  MoveL 707 to (-1326.52, 133.69, -285.52) mm, rotated rx 0 ry 47.8 rz 84.75 deg; joints [-10.196, -86.438, 119.109, 34.441, 19.155, -37.06]
  MoveL 708 to (-1326.52, 139.05, -290.91) mm, rotated rx 0 ry 42.78 rz 82.49 deg; joints [-10.577, -86.69, 120.873, 54.085, 15.911, -54.797]
  MoveL 709 to (-1326.52, 145, -295.87) mm, rotated rx 0 ry 37.57 rz 79.59 deg; joints [-10.961, -86.687, 122.605, 80.895, 15.197, -79.11]
  MoveL 710 to (-1326.52, 151.65, -300.42) mm, rotated rx 0 ry 32.53 rz 76.01 deg; joints [-11.319, -86.401, 124.196, 105.031, 17.66, -100.073]
  MoveL 711 to (-1326.52, 159.08, -304.57) mm, rotated rx 0 ry 27.96 rz 71.68 deg; joints [-11.629, -85.86, 125.576, 120.71, 22.02, -111.85]
  MoveL 712 to (-1326.52, 167.44, -308.37) mm, rotated rx 0 ry 24.05 rz 66.65 deg; joints [-11.882, -85.127, 126.726, 130.104, 26.9, -116.621]
  MoveL 713 to (-1326.52, 176.82, -311.83) mm, rotated rx 0 ry 20.87 rz 61.02 deg; joints [-12.081, -84.273, 127.659, 135.936, 31.589, -117.213]
  MoveL 714 to (-1326.52, 187.35, -315) mm, rotated rx 0 ry 18.39 rz 55.01 deg; joints [-12.232, -83.355, 128.413, 139.778, 35.812, -115.407]
  MoveL 715 to (-1326.52, 199.25, -317.93) mm, rotated rx 0 ry 16.51 rz 48.84 deg; joints [-12.346, -82.397, 129.031, 142.477, 39.539, -112.288]
  MoveL 716 to (-1326.52, 212.75, -320.67) mm, rotated rx 0 ry 15.13 rz 42.79 deg; joints [-12.432, -81.406, 129.549, 144.477, 42.811, -108.587]
  MoveL 717 to (-1326.52, 228.02, -323.22) mm, rotated rx 0 ry 14.14 rz 37.16 deg; joints [-12.496, -80.381, 129.992, 146.027, 45.69, -104.838]
  MoveL 718 to (-1326.52, 236.37, -324.43) mm, rotated rx 0 ry 13.75 rz 34.56 deg; joints [-12.522, -79.853, 130.191, 146.684, 47.005, -103.062]
  MoveL 719 to (-1326.52, 245.24, -325.61) mm, rotated rx 0 ry 13.43 rz 32.12 deg; joints [-12.544, -79.311, 130.378, 147.28, 48.252, -101.393]
  MoveL 720 to (-1326.52, 254.64, -326.75) mm, rotated rx 0 ry 13.16 rz 29.86 deg; joints [-12.563, -78.754, 130.555, 147.826, 49.438, -99.851]
  MoveL 721 to (-1326.52, 264.6, -327.86) mm, rotated rx 0 ry 12.93 rz 27.78 deg; joints [-12.579, -78.179, 130.722, 148.331, 50.574, -98.447]
  MoveL 722 to (-1326.52, 275.13, -328.94) mm, rotated rx 0 ry 12.74 rz 25.87 deg; joints [-12.593, -77.584, 130.88, 148.801, 51.667, -97.189]
  MoveL 723 to (-1326.52, 286.26, -330) mm, rotated rx 0 ry 12.58 rz 24.13 deg; joints [-12.605, -76.967, 131.03, 149.244, 52.726, -96.078]
  MoveL 724 to (-1326.52, 286.26, -330) mm, rotated rx 0 ry 12.58 rz 24.13 deg; joints [-12.605, -76.967, 131.03, 149.244, 52.726, -96.078]
  MoveL 725 to (-1327.33, 298.07, -330.87) mm, rotated rx 0 ry 12.44 rz 22.54 deg; joints [-12.64, -76.309, 131.156, 149.627, 53.768, -95.074]
  MoveL 726 to (-1329.7, 309.72, -331.34) mm, rotated rx 0 ry 12.34 rz 21.17 deg; joints [-12.72, -75.646, 131.236, 149.894, 54.732, -94.208]
  MoveL 727 to (-1333.52, 320.91, -331.42) mm, rotated rx 0 ry 12.28 rz 20.03 deg; joints [-12.842, -74.994, 131.269, 150.052, 55.607, -93.471]
  MoveL 728 to (-1338.76, 331.5, -331.11) mm, rotated rx 0 ry 12.24 rz 19.08 deg; joints [-13.005, -74.361, 131.258, 150.106, 56.395, -92.839]
  MoveL 729 to (-1345.4, 341.17, -330.42) mm, rotated rx 0 ry 12.22 rz 18.3 deg; joints [-13.209, -73.762, 131.202, 150.06, 57.086, -92.294]
  MoveL 730 to (-1349.24, 345.58, -329.93) mm, rotated rx 0 ry 12.22 rz 17.97 deg; joints [-13.326, -73.48, 131.157, 149.999, 57.393, -92.047]
  MoveL 731 to (-1353.42, 349.63, -329.34) mm, rotated rx 0 ry 12.23 rz 17.68 deg; joints [-13.452, -73.213, 131.101, 149.912, 57.67, -91.816]
  MoveL 732 to (-1357.93, 353.26, -328.64) mm, rotated rx 0 ry 12.24 rz 17.43 deg; joints [-13.588, -72.964, 131.033, 149.799, 57.915, -91.597]
  MoveL 733 to (-1362.76, 356.39, -327.84) mm, rotated rx 0 ry 12.26 rz 17.22 deg; joints [-13.733, -72.737, 130.954, 149.66, 58.125, -91.39]
  MoveL 734 to (-1367.87, 358.95, -326.94) mm, rotated rx 0 ry 12.28 rz 17.05 deg; joints [-13.886, -72.537, 130.864, 149.495, 58.297, -91.193]
  MoveL 735 to (-1373.23, 360.86, -325.95) mm, rotated rx 0 ry 12.31 rz 16.92 deg; joints [-14.045, -72.369, 130.763, 149.304, 58.425, -91.006]
  MoveL 736 to (-1378.75, 362.03, -324.87) mm, rotated rx 0 ry 12.34 rz 16.84 deg; joints [-14.209, -72.236, 130.653, 149.089, 58.506, -90.83]
  MoveL 737 to (-1384.36, 362.38, -323.72) mm, rotated rx 0 ry 12.37 rz 16.79 deg; joints [-14.374, -72.145, 130.535, 148.852, 58.536, -90.665]
  MoveL 738 to (-1389.91, 361.87, -322.52) mm, rotated rx 0 ry 12.41 rz 16.8 deg; joints [-14.537, -72.098, 130.412, 148.598, 58.514, -90.514]
  MoveL 739 to (-1395.3, 360.5, -321.29) mm, rotated rx 0 ry 12.45 rz 16.85 deg; joints [-14.694, -72.097, 130.286, 148.332, 58.439, -90.381]
  MoveL 740 to (-1400.38, 358.32, -320.08) mm, rotated rx 0 ry 12.5 rz 16.95 deg; joints [-14.842, -72.14, 130.161, 148.059, 58.315, -90.267]
  MoveL 741 to (-1405.09, 355.4, -318.88) mm, rotated rx 0 ry 12.54 rz 17.09 deg; joints [-14.978, -72.226, 130.038, 147.784, 58.145, -90.176]
  MoveL 742 to (-1409.35, 351.85, -317.74) mm, rotated rx 0 ry 12.59 rz 17.28 deg; joints [-15.1, -72.349, 129.919, 147.511, 57.935, -90.111]
  MoveL 743 to (-1413.12, 347.77, -316.66) mm, rotated rx 0 ry 12.64 rz 17.51 deg; joints [-15.207, -72.505, 129.806, 147.245, 57.69, -90.073]
  MoveL 744 to (-1416.4, 343.25, -315.65) mm, rotated rx 0 ry 12.68 rz 17.77 deg; joints [-15.3, -72.689, 129.699, 146.986, 57.416, -90.065]
  MoveL 745 to (-1419.19, 338.39, -314.72) mm, rotated rx 0 ry 12.73 rz 18.07 deg; joints [-15.378, -72.896, 129.599, 146.736, 57.115, -90.087]
  MoveL 746 to (-1421.51, 333.27, -313.86) mm, rotated rx 0 ry 12.77 rz 18.41 deg; joints [-15.442, -73.123, 129.506, 146.495, 56.793, -90.142]
  MoveL 747 to (-1423.36, 327.94, -313.08) mm, rotated rx 0 ry 12.82 rz 18.78 deg; joints [-15.493, -73.367, 129.419, 146.264, 56.451, -90.232]
  MoveL 748 to (-1425.75, 316.92, -311.73) mm, rotated rx 0 ry 12.91 rz 19.64 deg; joints [-15.555, -73.892, 129.266, 145.831, 55.716, -90.518]
  MoveL 749 to (-1426.52, 305.59, -310.67) mm, rotated rx 0 ry 13 rz 20.66 deg; joints [-15.569, -74.457, 129.137, 145.433, 54.917, -90.961]
  MoveL 750 to (-1426.52, 305.59, -310.67) mm, rotated rx 0 ry 13 rz 20.66 deg; joints [-15.569, -74.457, 129.137, 145.433, 54.917, -90.961]
  MoveL 751 to (-1426.52, 292.69, -309.58) mm, rotated rx 0 ry 13.12 rz 22.01 deg; joints [-15.558, -75.118, 128.996, 144.979, 53.948, -91.637]
  MoveL 752 to (-1426.52, 280.46, -308.47) mm, rotated rx 0 ry 13.26 rz 23.51 deg; joints [-15.546, -75.751, 128.846, 144.501, 52.958, -92.447]
  MoveL 753 to (-1426.52, 268.86, -307.34) mm, rotated rx 0 ry 13.42 rz 25.16 deg; joints [-15.532, -76.359, 128.689, 143.995, 51.943, -93.394]
  MoveL 754 to (-1426.52, 257.88, -306.18) mm, rotated rx 0 ry 13.61 rz 26.98 deg; joints [-15.516, -76.944, 128.524, 143.455, 50.894, -94.481]
  MoveL 755 to (-1426.52, 247.5, -304.99) mm, rotated rx 0 ry 13.83 rz 28.98 deg; joints [-15.498, -77.508, 128.349, 142.875, 49.804, -95.706]
  MoveL 756 to (-1426.52, 237.7, -303.77) mm, rotated rx 0 ry 14.1 rz 31.15 deg; joints [-15.477, -78.055, 128.165, 142.246, 48.666, -97.065]
  MoveL 757 to (-1426.52, 228.44, -302.52) mm, rotated rx 0 ry 14.42 rz 33.5 deg; joints [-15.453, -78.585, 127.971, 141.559, 47.47, -98.545]
  MoveL 758 to (-1426.52, 219.71, -301.22) mm, rotated rx 0 ry 14.79 rz 36.02 deg; joints [-15.425, -79.103, 127.764, 140.801, 46.207, -100.128]
  MoveL 759 to (-1426.52, 203.75, -298.5) mm, rotated rx 0 ry 15.77 rz 41.51 deg; joints [-15.356, -80.104, 127.306, 139.011, 43.445, -103.484]
  MoveL 760 to (-1426.52, 189.63, -295.6) mm, rotated rx 0 ry 17.13 rz 47.47 deg; joints [-15.264, -81.069, 126.774, 136.704, 40.309, -106.789]
  MoveL 761 to (-1426.52, 177.19, -292.48) mm, rotated rx 0 ry 18.98 rz 53.62 deg; joints [-15.142, -82.002, 126.14, 133.606, 36.747, -109.502]
  MoveL 762 to (-1426.52, 166.2, -289.11) mm, rotated rx 0 ry 21.44 rz 59.69 deg; joints [-14.98, -82.892, 125.371, 129.255, 32.744, -110.863]
  MoveL 763 to (-1426.52, 156.45, -285.45) mm, rotated rx 0 ry 24.62 rz 65.42 deg; joints [-14.766, -83.716, 124.423, 122.809, 28.363, -109.781]
  MoveL 764 to (-1426.52, 147.8, -281.45) mm, rotated rx 0 ry 28.53 rz 70.58 deg; joints [-14.491, -84.42, 123.258, 112.872, 23.92, -104.636]
  MoveL 765 to (-1426.52, 140.12, -277.09) mm, rotated rx 0 ry 33.13 rz 75.06 deg; joints [-14.153, -84.935, 121.859, 97.493, 20.141, -93.356]
  MoveL 766 to (-1426.52, 133.29, -272.32) mm, rotated rx 0 ry 38.23 rz 78.81 deg; joints [-13.758, -85.198, 120.243, 76.054, 18.22, -75.297]
  MoveL 767 to (-1426.52, 127.2, -267.12) mm, rotated rx 0 ry 43.54 rz 81.87 deg; joints [-13.328, -85.179, 118.475, 53.313, 19.065, -55.259]
  MoveL 768 to (-1426.52, 121.74, -261.48) mm, rotated rx 0 ry 48.7 rz 84.29 deg; joints [-12.895, -84.901, 116.664, 35.753, 22.135, -39.8]
  MoveL 769 to (-1426.52, 116.79, -255.37) mm, rotated rx 0 ry 53.41 rz 86.16 deg; joints [-12.491, -84.434, 114.915, 24.338, 26.12, -29.975]
  MoveL 770 to (-1426.52, 112.26, -248.79) mm, rotated rx 0 ry 57.46 rz 87.56 deg; joints [-12.139, -83.866, 113.312, 17.209, 30.068, -24.015]
  MoveL 771 to (-1426.52, 104.19, -234.49) mm, rotated rx 0 ry 63.1 rz 89.23 deg; joints [-11.637, -82.74, 110.762, 10.074, 36.099, -18.238]
  MoveL 772 to (-1426.52, 100.41, -226.7) mm, rotated rx 0 ry 64.85 rz 89.65 deg; joints [-11.475, -82.248, 109.781, 8.382, 38.115, -16.881]
  MoveL 773 to (-1426.52, 96.59, -218.35) mm, rotated rx 0 ry 65.93 rz 89.83 deg; joints [-11.368, -81.826, 108.976, 7.504, 39.473, -16.142]
  MoveL 774 to (-1426.52, 92.67, -209.5) mm, rotated rx 0 ry 66.26 rz 89.73 deg; joints [-11.328, -81.505, 108.379, 7.43, 40.076, -15.986]
  MoveL 775 to (-1426.52, 89.09, -201.31) mm, rotated rx 0 ry 66.5 rz 89.64 deg; joints [-11.292, -81.216, 107.846, 7.394, 40.567, -15.869]
  MoveL 776 to (-1426.52, 82.11, -185.13) mm, rotated rx 0 ry 66.74 rz 89.47 deg; joints [-11.23, -80.682, 106.868, 7.427, 41.278, -15.73]
  MoveL 777 to (-1426.52, 78.05, -175.71) mm, rotated rx 0 ry 66.67 rz 89.37 deg; joints [-11.199, -80.409, 106.368, 7.531, 41.456, -15.723]
  MoveL 778 to (-1426.52, 75.74, -170.35) mm, rotated rx 0 ry 66.62 rz 89.32 deg; joints [-11.182, -80.256, 106.087, 7.589, 41.545, -15.719]
  MoveL 779 to (-1426.52, 73.19, -164.48) mm, rotated rx 0 ry 66.56 rz 89.27 deg; joints [-11.162, -80.09, 105.78, 7.651, 41.634, -15.714]
  MoveL 780 to (-1426.52, 67.8, -152.08) mm, rotated rx 0 ry 66.4 rz 89.18 deg; joints [-11.12, -79.742, 105.137, 7.77, 41.796, -15.701]
  MoveL 781 to (-1426.52, 62.1, -139.11) mm, rotated rx 0 ry 66.22 rz 89.1 deg; joints [-11.073, -79.384, 104.471, 7.875, 41.938, -15.676]
  MoveL 782 to (-1426.52, 49.92, -111.76) mm, rotated rx 0 ry 65.77 rz 89.01 deg; joints [-10.966, -78.642, 103.075, 8.006, 42.161, -15.581]
  MoveL 783 to (-1426.52, 36.86, -83.09) mm, rotated rx 0 ry 65.22 rz 89.05 deg; joints [-10.84, -77.882, 101.625, 7.994, 42.293, -15.408]
  MoveL 784 to (-1426.52, 36.86, -83.09) mm, rotated rx 0 ry 65.22 rz 89.05 deg; joints [-10.84, -77.882, 101.625, 7.994, 42.293, -15.408]
  MoveL 785 to (-1427.42, 32.64, -73.95) mm, rotated rx 0 ry 65.02 rz 89.09 deg; joints [-10.818, -77.638, 101.16, 7.969, 42.309, -15.367]
  MoveL 786 to (-1430.11, 28.53, -65.1) mm, rotated rx 0 ry 64.81 rz 89.15 deg; joints [-10.839, -77.393, 100.7, 7.957, 42.303, -15.383]
  MoveL 787 to (-1434.53, 24.7, -56.86) mm, rotated rx 0 ry 64.58 rz 89.22 deg; joints [-10.904, -77.157, 100.265, 7.966, 42.269, -15.46]
  MoveL 788 to (-1440.57, 21.28, -49.53) mm, rotated rx 0 ry 64.34 rz 89.3 deg; joints [-11.012, -76.937, 99.869, 8.005, 42.207, -15.601]
  MoveL 789 to (-1444.15, 19.76, -46.29) mm, rotated rx 0 ry 64.22 rz 89.33 deg; joints [-11.081, -76.836, 99.691, 8.038, 42.166, -15.697]
  MoveL 790 to (-1448.06, 18.41, -43.41) mm, rotated rx 0 ry 64.1 rz 89.37 deg; joints [-11.16, -76.742, 99.529, 8.08, 42.121, -15.807]
  MoveL 791 to (-1452.27, 17.23, -40.89) mm, rotated rx 0 ry 63.98 rz 89.4 deg; joints [-11.248, -76.656, 99.384, 8.131, 42.072, -15.932]
  MoveL 792 to (-1456.75, 16.23, -38.77) mm, rotated rx 0 ry 63.87 rz 89.43 deg; joints [-11.344, -76.578, 99.256, 8.192, 42.022, -16.072]
  MoveL 793 to (-1461.45, 15.45, -37.08) mm, rotated rx 0 ry 63.77 rz 89.45 deg; joints [-11.448, -76.509, 99.148, 8.261, 41.973, -16.224]
  MoveL 794 to (-1466.32, 14.88, -35.84) mm, rotated rx 0 ry 63.69 rz 89.47 deg; joints [-11.559, -76.449, 99.06, 8.339, 41.926, -16.386]
  MoveL 795 to (-1471.31, 14.55, -35.07) mm, rotated rx 0 ry 63.61 rz 89.49 deg; joints [-11.675, -76.4, 98.993, 8.423, 41.885, -16.557]
  MoveL 796 to (-1476.37, 14.45, -34.79) mm, rotated rx 0 ry 63.56 rz 89.5 deg; joints [-11.795, -76.361, 98.947, 8.511, 41.851, -16.734]
  MoveL 797 to (-1481.42, 14.59, -34.98) mm, rotated rx 0 ry 63.52 rz 89.5 deg; joints [-11.917, -76.332, 98.923, 8.603, 41.826, -16.913]
  MoveL 798 to (-1486.42, 14.98, -35.66) mm, rotated rx 0 ry 63.5 rz 89.5 deg; joints [-12.041, -76.313, 98.919, 8.695, 41.812, -17.093]
  MoveL 799 to (-1491.31, 15.59, -36.81) mm, rotated rx 0 ry 63.5 rz 89.49 deg; joints [-12.164, -76.305, 98.937, 8.786, 41.809, -17.271]
  MoveL 800 to (-1496.04, 16.43, -38.41) mm, rotated rx 0 ry 63.53 rz 89.48 deg; joints [-12.286, -76.308, 98.974, 8.872, 41.817, -17.443]
  MoveL 801 to (-1500.54, 17.49, -40.44) mm, rotated rx 0 ry 63.57 rz 89.46 deg; joints [-12.405, -76.321, 99.032, 8.953, 41.837, -17.608]
  MoveL 802 to (-1504.79, 18.74, -42.88) mm, rotated rx 0 ry 63.64 rz 89.45 deg; joints [-12.52, -76.343, 99.108, 9.026, 41.868, -17.763]
  MoveL 803 to (-1508.74, 20.17, -45.7) mm, rotated rx 0 ry 63.72 rz 89.43 deg; joints [-12.629, -76.376, 99.202, 9.09, 41.909, -17.907]
  MoveL 804 to (-1512.34, 21.76, -48.86) mm, rotated rx 0 ry 63.82 rz 89.41 deg; joints [-12.731, -76.419, 99.313, 9.143, 41.959, -18.037]
  MoveL 805 to (-1518.45, 25.35, -56.07) mm, rotated rx 0 ry 64.07 rz 89.37 deg; joints [-12.914, -76.531, 99.582, 9.215, 42.078, -18.255]
  MoveL 806 to (-1522.9, 29.33, -64.21) mm, rotated rx 0 ry 64.37 rz 89.34 deg; joints [-13.06, -76.677, 99.906, 9.238, 42.212, -18.409]
  MoveL 807 to (-1525.62, 33.55, -73) mm, rotated rx 0 ry 64.69 rz 89.32 deg; joints [-13.167, -76.855, 100.276, 9.214, 42.346, -18.499]
  MoveL 808 to (-1526.52, 37.84, -82.11) mm, rotated rx 0 ry 65.01 rz 89.31 deg; joints [-13.231, -77.057, 100.68, 9.149, 42.468, -18.526]
  MoveL 809 to (-1526.52, 37.84, -82.11) mm, rotated rx 0 ry 65.01 rz 89.31 deg; joints [-13.231, -77.057, 100.68, 9.149, 42.468, -18.526]
  MoveL 810 to (-1526.52, 47.5, -103.17) mm, rotated rx 0 ry 65.71 rz 89.33 deg; joints [-13.324, -77.556, 101.645, 8.921, 42.682, -18.502]
  MoveL 811 to (-1526.52, 56.25, -122.84) mm, rotated rx 0 ry 66.32 rz 89.42 deg; joints [-13.404, -78.037, 102.559, 8.647, 42.81, -18.454]
  MoveL 812 to (-1526.52, 60.26, -132.03) mm, rotated rx 0 ry 66.58 rz 89.48 deg; joints [-13.44, -78.266, 102.989, 8.501, 42.847, -18.424]
  MoveL 813 to (-1526.52, 64, -140.72) mm, rotated rx 0 ry 66.81 rz 89.54 deg; joints [-13.472, -78.486, 103.4, 8.354, 42.866, -18.392]
  MoveL 814 to (-1526.52, 67.48, -148.88) mm, rotated rx 0 ry 67.02 rz 89.62 deg; joints [-13.502, -78.695, 103.788, 8.209, 42.869, -18.359]
  MoveL 815 to (-1526.52, 70.67, -156.45) mm, rotated rx 0 ry 67.2 rz 89.69 deg; joints [-13.529, -78.893, 104.152, 8.071, 42.857, -18.328]
  MoveL 816 to (-1526.52, 73.57, -163.37) mm, rotated rx 0 ry 67.35 rz 89.76 deg; joints [-13.554, -79.076, 104.488, 7.944, 42.831, -18.299]
  MoveL 817 to (-1526.52, 76.11, -169.48) mm, rotated rx 0 ry 67.47 rz 89.83 deg; joints [-13.576, -79.24, 104.788, 7.831, 42.795, -18.276]
  MoveL 818 to (-1526.52, 78.33, -174.85) mm, rotated rx 0 ry 67.57 rz 89.89 deg; joints [-13.595, -79.386, 105.054, 7.733, 42.751, -18.256]
  MoveL 819 to (-1526.52, 80.27, -179.57) mm, rotated rx 0 ry 67.64 rz 89.95 deg; joints [-13.612, -79.516, 105.291, 7.648, 42.703, -18.241]
  MoveL 820 to (-1526.52, 83.53, -187.5) mm, rotated rx 0 ry 67.69 rz 90.03 deg; joints [-13.646, -79.749, 105.715, 7.574, 42.539, -18.265]
  MoveL 821 to (-1526.52, 86.29, -194.12) mm, rotated rx 0 ry 67.02 rz 89.88 deg; joints [-13.734, -80.058, 106.289, 8.173, 41.697, -18.757]
  MoveL 822 to (-1526.52, 91.81, -206.5) mm, rotated rx 0 ry 64.7 rz 89.27 deg; joints [-13.991, -80.786, 107.701, 10.471, 39.058, -20.565]
  MoveL 823 to (-1526.52, 98.21, -218.93) mm, rotated rx 0 ry 60.41 rz 87.95 deg; joints [-14.424, -81.724, 109.719, 15.653, 34.584, -24.637]
  MoveL 824 to (-1526.52, 105.6, -230.44) mm, rotated rx 0 ry 53.86 rz 85.6 deg; joints [-15.056, -82.709, 112.358, 26.575, 28.443, -33.527]
  MoveL 825 to (-1526.52, 114.25, -240.61) mm, rotated rx 0 ry 45.56 rz 81.92 deg; joints [-15.822, -83.387, 115.364, 48.173, 22.695, -51.859]
  MoveL 826 to (-1526.52, 119.2, -245.22) mm, rotated rx 0 ry 41.11 rz 79.47 deg; joints [-16.214, -83.494, 116.871, 63.803, 21.291, -65.277]
  MoveL 827 to (-1526.52, 124.65, -249.52) mm, rotated rx 0 ry 36.73 rz 76.56 deg; joints [-16.586, -83.412, 118.296, 80.496, 21.535, -79.316]
  MoveL 828 to (-1526.52, 130.66, -253.54) mm, rotated rx 0 ry 32.61 rz 73.16 deg; joints [-16.922, -83.144, 119.591, 95.345, 23.343, -91.039]
  MoveL 829 to (-1526.52, 137.32, -257.28) mm, rotated rx 0 ry 28.87 rz 69.28 deg; joints [-17.213, -82.716, 120.73, 106.89, 26.189, -98.976]
  MoveL 830 to (-1526.52, 144.69, -260.76) mm, rotated rx 0 ry 25.62 rz 64.95 deg; joints [-17.456, -82.164, 121.708, 115.314, 29.5, -103.343]
  MoveL 831 to (-1526.52, 152.84, -264.01) mm, rotated rx 0 ry 22.89 rz 60.24 deg; joints [-17.654, -81.527, 122.535, 121.4, 32.877, -104.997]
  MoveL 832 to (-1526.52, 161.84, -267.04) mm, rotated rx 0 ry 20.66 rz 55.29 deg; joints [-17.812, -80.836, 123.232, 125.859, 36.096, -104.774]
  MoveL 833 to (-1526.52, 171.81, -269.89) mm, rotated rx 0 ry 18.87 rz 50.22 deg; joints [-17.937, -80.11, 123.824, 129.212, 39.065, -103.338]
  MoveL 834 to (-1526.52, 182.89, -272.57) mm, rotated rx 0 ry 17.48 rz 45.21 deg; joints [-18.036, -79.358, 124.334, 131.806, 41.764, -101.194]
  MoveL 835 to (-1526.52, 195.16, -275.1) mm, rotated rx 0 ry 16.4 rz 40.41 deg; joints [-18.114, -78.583, 124.779, 133.865, 44.197, -98.73]
  MoveL 836 to (-1526.52, 208.73, -277.5) mm, rotated rx 0 ry 15.59 rz 35.95 deg; joints [-18.176, -77.783, 125.172, 135.54, 46.392, -96.234]
  MoveL 837 to (-1526.52, 223.7, -279.77) mm, rotated rx 0 ry 14.97 rz 31.92 deg; joints [-18.226, -76.953, 125.526, 136.938, 48.382, -93.902]
  MoveL 838 to (-1526.52, 240.17, -281.94) mm, rotated rx 0 ry 14.51 rz 28.35 deg; joints [-18.266, -76.083, 125.848, 138.132, 50.207, -91.852]
  MoveL 839 to (-1526.52, 258.24, -284.02) mm, rotated rx 0 ry 14.16 rz 25.27 deg; joints [-18.298, -75.165, 126.143, 139.176, 51.902, -90.143]
  MoveL 840 to (-1526.52, 278.01, -286.02) mm, rotated rx 0 ry 13.89 rz 22.63 deg; joints [-18.325, -74.187, 126.415, 140.108, 53.502, -88.795]
  MoveL 841 to (-1526.52, 299.59, -287.96) mm, rotated rx 0 ry 13.68 rz 20.4 deg; joints [-18.346, -73.138, 126.665, 140.955, 55.037, -87.8]
  MoveL 842 to (-1526.52, 299.59, -287.96) mm, rotated rx 0 ry 13.68 rz 20.4 deg; joints [-18.346, -73.138, 126.665, 140.955, 55.037, -87.8]
  MoveL 843 to (-1527.37, 311.74, -288.77) mm, rotated rx 0 ry 13.59 rz 19.37 deg; joints [-18.379, -72.538, 126.766, 141.34, 55.834, -87.383]
  MoveL 844 to (-1529.86, 323.82, -289.14) mm, rotated rx 0 ry 13.53 rz 18.48 deg; joints [-18.455, -71.918, 126.813, 141.622, 56.591, -87.018]
  MoveL 845 to (-1533.91, 335.46, -289.08) mm, rotated rx 0 ry 13.49 rz 17.71 deg; joints [-18.572, -71.295, 126.806, 141.802, 57.291, -86.702]
  MoveL 846 to (-1539.39, 346.28, -288.61) mm, rotated rx 0 ry 13.47 rz 17.08 deg; joints [-18.725, -70.691, 126.747, 141.88, 57.918, -86.426]
  MoveL 847 to (-1546.08, 355.9, -287.74) mm, rotated rx 0 ry 13.47 rz 16.58 deg; joints [-18.91, -70.128, 126.64, 141.862, 58.457, -86.177]
  MoveL 848 to (-1553.86, 364.07, -286.5) mm, rotated rx 0 ry 13.48 rz 16.18 deg; joints [-19.121, -69.618, 126.489, 141.755, 58.903, -85.943]
  MoveL 849 to (-1558.2, 367.6, -285.74) mm, rotated rx 0 ry 13.49 rz 16.02 deg; joints [-19.238, -69.384, 126.396, 141.667, 59.092, -85.824]
  MoveL 850 to (-1562.83, 370.68, -284.87) mm, rotated rx 0 ry 13.51 rz 15.89 deg; joints [-19.362, -69.166, 126.292, 141.556, 59.256, -85.702]
  MoveL 851 to (-1567.74, 373.25, -283.9) mm, rotated rx 0 ry 13.53 rz 15.77 deg; joints [-19.493, -68.968, 126.176, 141.42, 59.393, -85.576]
  MoveL 852 to (-1572.89, 375.23, -282.84) mm, rotated rx 0 ry 13.56 rz 15.69 deg; joints [-19.63, -68.795, 126.05, 141.261, 59.497, -85.445]
  MoveL 853 to (-1578.23, 376.53, -281.68) mm, rotated rx 0 ry 13.59 rz 15.63 deg; joints [-19.77, -68.65, 125.913, 141.078, 59.568, -85.308]
  MoveL 854 to (-1583.66, 377.08, -280.45) mm, rotated rx 0 ry 13.62 rz 15.6 deg; joints [-19.913, -68.54, 125.769, 140.874, 59.6, -85.166]
  MoveL 855 to (-1589.12, 376.81, -279.16) mm, rotated rx 0 ry 13.66 rz 15.6 deg; joints [-20.054, -68.466, 125.62, 140.65, 59.593, -85.02]
  MoveL 856 to (-1594.43, 375.72, -277.85) mm, rotated rx 0 ry 13.7 rz 15.63 deg; joints [-20.192, -68.433, 125.468, 140.412, 59.546, -84.874]
  MoveL 857 to (-1599.51, 373.81, -276.53) mm, rotated rx 0 ry 13.73 rz 15.69 deg; joints [-20.322, -68.44, 125.318, 140.164, 59.459, -84.729]
  MoveL 858 to (-1604.27, 371.14, -275.23) mm, rotated rx 0 ry 13.78 rz 15.78 deg; joints [-20.443, -68.487, 125.171, 139.909, 59.335, -84.591]
  MoveL 859 to (-1608.59, 367.81, -273.98) mm, rotated rx 0 ry 13.82 rz 15.91 deg; joints [-20.552, -68.57, 125.031, 139.655, 59.178, -84.462]
  MoveL 860 to (-1612.45, 363.91, -272.8) mm, rotated rx 0 ry 13.86 rz 16.05 deg; joints [-20.649, -68.686, 124.9, 139.403, 58.993, -84.347]
  MoveL 861 to (-1615.83, 359.54, -271.7) mm, rotated rx 0 ry 13.9 rz 16.23 deg; joints [-20.733, -68.831, 124.777, 139.156, 58.783, -84.246]
  MoveL 862 to (-1618.72, 354.79, -270.68) mm, rotated rx 0 ry 13.93 rz 16.43 deg; joints [-20.804, -68.999, 124.665, 138.916, 58.553, -84.164]
  MoveL 863 to (-1621.12, 349.75, -269.75) mm, rotated rx 0 ry 13.97 rz 16.66 deg; joints [-20.862, -69.189, 124.562, 138.684, 58.304, -84.102]
  MoveL 864 to (-1623.06, 344.48, -268.91) mm, rotated rx 0 ry 14.01 rz 16.91 deg; joints [-20.908, -69.396, 124.47, 138.461, 58.041, -84.06]
  MoveL 865 to (-1625.65, 333.23, -267.46) mm, rotated rx 0 ry 14.08 rz 17.49 deg; joints [-20.966, -69.862, 124.31, 138.032, 57.464, -84.048]
  MoveL 866 to (-1626.52, 321.21, -266.33) mm, rotated rx 0 ry 14.16 rz 18.2 deg; joints [-20.979, -70.392, 124.185, 137.626, 56.819, -84.145]
  MoveL 867 to (-1626.52, 321.21, -266.33) mm, rotated rx 0 ry 14.16 rz 18.2 deg; joints [-20.979, -70.392, 124.185, 137.626, 56.819, -84.145]
  MoveL 868 to (-1626.52, 308.51, -265.3) mm, rotated rx 0 ry 14.24 rz 19.05 deg; joints [-20.968, -70.968, 124.067, 137.204, 56.102, -84.351]
  MoveL 869 to (-1626.52, 296.33, -264.27) mm, rotated rx 0 ry 14.33 rz 20 deg; joints [-20.957, -71.522, 123.943, 136.766, 55.379, -84.636]
  MoveL 870 to (-1626.52, 273.48, -262.16) mm, rotated rx 0 ry 14.54 rz 22.17 deg; joints [-20.932, -72.569, 123.678, 135.832, 53.899, -85.456]
  MoveL 871 to (-1626.52, 252.55, -259.98) mm, rotated rx 0 ry 14.81 rz 24.75 deg; joints [-20.901, -73.543, 123.389, 134.802, 52.354, -86.625]
  MoveL 872 to (-1626.52, 233.44, -257.72) mm, rotated rx 0 ry 15.17 rz 27.8 deg; joints [-20.865, -74.455, 123.076, 133.643, 50.712, -88.152]
  MoveL 873 to (-1626.52, 216.04, -255.36) mm, rotated rx 0 ry 15.64 rz 31.32 deg; joints [-20.821, -75.316, 122.735, 132.312, 48.941, -90.016]
  MoveL 874 to (-1626.52, 200.24, -252.89) mm, rotated rx 0 ry 16.27 rz 35.34 deg; joints [-20.767, -76.137, 122.36, 130.748, 47.004, -92.157]
  MoveL 875 to (-1626.52, 185.94, -250.28) mm, rotated rx 0 ry 17.11 rz 39.81 deg; joints [-20.698, -76.925, 121.942, 128.866, 44.866, -94.451]
  MoveL 876 to (-1626.52, 173.02, -247.52) mm, rotated rx 0 ry 18.23 rz 44.64 deg; joints [-20.613, -77.687, 121.471, 126.548, 42.493, -96.692]
  MoveL 877 to (-1626.52, 161.39, -244.6) mm, rotated rx 0 ry 19.68 rz 49.72 deg; joints [-20.504, -78.425, 120.93, 123.624, 39.866, -98.576]
  MoveL 878 to (-1626.52, 150.93, -241.5) mm, rotated rx 0 ry 21.55 rz 54.86 deg; joints [-20.366, -79.134, 120.3, 119.849, 36.989, -99.688]
  MoveL 879 to (-1626.52, 141.5, -238.19) mm, rotated rx 0 ry 23.89 rz 59.92 deg; joints [-20.191, -79.804, 119.556, 114.856, 33.904, -99.495]
  MoveL 880 to (-1626.52, 132.99, -234.63) mm, rotated rx 0 ry 26.78 rz 64.73 deg; joints [-19.971, -80.415, 118.671, 108.116, 30.733, -97.32]
  MoveL 881 to (-1626.52, 125.3, -230.8) mm, rotated rx 0 ry 30.22 rz 69.17 deg; joints [-19.698, -80.932, 117.624, 99.007, 27.745, -92.406]
  MoveL 882 to (-1626.52, 118.38, -226.68) mm, rotated rx 0 ry 34.16 rz 73.14 deg; joints [-19.371, -81.315, 116.403, 87.049, 25.383, -84.187]
  MoveL 883 to (-1626.52, 112.13, -222.25) mm, rotated rx 0 ry 38.51 rz 76.61 deg; joints [-18.992, -81.524, 115.019, 72.575, 24.192, -72.961]
  MoveL 884 to (-1626.52, 106.48, -217.48) mm, rotated rx 0 ry 43.09 rz 79.58 deg; joints [-18.573, -81.536, 113.504, 57.318, 24.55, -60.465]
  MoveL 885 to (-1626.52, 101.38, -212.38) mm, rotated rx 0 ry 47.69 rz 82.07 deg; joints [-18.135, -81.354, 111.919, 43.63, 26.369, -49.076]
  MoveL 886 to (-1626.52, 96.75, -206.92) mm, rotated rx 0 ry 52.08 rz 84.12 deg; joints [-17.703, -81.008, 110.335, 32.799, 29.146, -40.123]
  MoveL 887 to (-1626.52, 88.62, -194.9) mm, rotated rx 0 ry 59.56 rz 87.1 deg; joints [-16.934, -80.028, 107.418, 19.074, 35.391, -29.085]
  MoveL 888 to (-1626.52, 81.49, -181.31) mm, rotated rx 0 ry 64.57 rz 88.9 deg; joints [-16.371, -79.014, 105.128, 12.296, 40.273, -23.861]
  MoveL 889 to (-1626.52, 74.87, -166.4) mm, rotated rx 0 ry 67.16 rz 89.83 deg; joints [-16.019, -78.201, 103.51, 9.253, 43.065, -21.546]
  MoveL 890 to (-1626.52, 68.39, -150.56) mm, rotated rx 0 ry 68 rz 90.15 deg; joints [-15.826, -77.601, 102.379, 8.221, 44.24, -20.689]
  MoveL 891 to (-1626.52, 65.03, -142.31) mm, rotated rx 0 ry 67.71 rz 90.05 deg; joints [-15.797, -77.402, 102.014, 8.453, 44.16, -20.775]
  MoveL 892 to (-1626.52, 61.28, -133.25) mm, rotated rx 0 ry 67.37 rz 89.95 deg; joints [-15.765, -77.189, 101.619, 8.708, 44.048, -20.871]
  MoveL 893 to (-1626.52, 57.11, -123.34) mm, rotated rx 0 ry 66.97 rz 89.86 deg; joints [-15.729, -76.961, 101.193, 8.984, 43.9, -20.977]
  MoveL 894 to (-1626.52, 52.53, -112.68) mm, rotated rx 0 ry 66.52 rz 89.77 deg; joints [-15.689, -76.722, 100.741, 9.275, 43.712, -21.091]
  MoveL 895 to (-1626.52, 47.54, -101.34) mm, rotated rx 0 ry 66.01 rz 89.69 deg; joints [-15.645, -76.473, 100.266, 9.574, 43.484, -21.21]
  MoveL 896 to (-1626.52, 42.16, -89.4) mm, rotated rx 0 ry 65.45 rz 89.63 deg; joints [-15.597, -76.218, 99.772, 9.875, 43.212, -21.332]
  MoveL 897 to (-1626.52, 42.16, -89.4) mm, rotated rx 0 ry 65.45 rz 89.63 deg; joints [-15.597, -76.218, 99.772, 9.875, 43.212, -21.332]
  MoveL 898 to (-1627.42, 37.95, -80.26) mm, rotated rx 0 ry 65.01 rz 89.6 deg; joints [-15.58, -76.018, 99.386, 10.103, 42.987, -21.449]
  MoveL 899 to (-1630.12, 33.81, -71.42) mm, rotated rx 0 ry 64.56 rz 89.59 deg; joints [-15.604, -75.809, 98.994, 10.333, 42.76, -21.614]
  MoveL 900 to (-1634.55, 29.9, -63.23) mm, rotated rx 0 ry 64.13 rz 89.6 deg; joints [-15.67, -75.6, 98.611, 10.567, 42.535, -21.827]
  MoveL 901 to (-1640.62, 26.39, -55.96) mm, rotated rx 0 ry 63.72 rz 89.61 deg; joints [-15.777, -75.397, 98.249, 10.804, 42.321, -22.086]
  MoveL 902 to (-1644.21, 24.83, -52.77) mm, rotated rx 0 ry 63.53 rz 89.63 deg; joints [-15.845, -75.299, 98.081, 10.922, 42.222, -22.232]
  MoveL 903 to (-1648.13, 23.43, -49.93) mm, rotated rx 0 ry 63.35 rz 89.64 deg; joints [-15.923, -75.206, 97.923, 11.039, 42.132, -22.385]
  MoveL 904 to (-1652.36, 22.21, -47.45) mm, rotated rx 0 ry 63.19 rz 89.65 deg; joints [-16.009, -75.117, 97.776, 11.153, 42.051, -22.546]
  MoveL 905 to (-1656.85, 21.18, -45.37) mm, rotated rx 0 ry 63.05 rz 89.67 deg; joints [-16.103, -75.032, 97.642, 11.264, 41.984, -22.711]
  MoveL 906 to (-1661.56, 20.37, -43.72) mm, rotated rx 0 ry 62.93 rz 89.68 deg; joints [-16.203, -74.954, 97.521, 11.369, 41.933, -22.879]
  MoveL 907 to (-1666.44, 19.78, -42.52) mm, rotated rx 0 ry 62.85 rz 89.69 deg; joints [-16.31, -74.881, 97.414, 11.465, 41.9, -23.047]
  MoveL 908 to (-1671.43, 19.43, -41.79) mm, rotated rx 0 ry 62.79 rz 89.7 deg; joints [-16.421, -74.816, 97.323, 11.552, 41.887, -23.212]
  MoveL 909 to (-1676.49, 19.32, -41.53) mm, rotated rx 0 ry 62.76 rz 89.71 deg; joints [-16.536, -74.757, 97.247, 11.626, 41.895, -23.371]
  MoveL 910 to (-1681.54, 19.46, -41.75) mm, rotated rx 0 ry 62.76 rz 89.72 deg; joints [-16.653, -74.706, 97.187, 11.684, 41.927, -23.521]
  MoveL 911 to (-1686.53, 19.84, -42.44) mm, rotated rx 0 ry 62.8 rz 89.73 deg; joints [-16.77, -74.663, 97.144, 11.726, 41.982, -23.659]
  MoveL 912 to (-1691.41, 20.46, -43.6) mm, rotated rx 0 ry 62.87 rz 89.73 deg; joints [-16.886, -74.629, 97.118, 11.749, 42.06, -23.783]
  MoveL 913 to (-1696.13, 21.3, -45.21) mm, rotated rx 0 ry 62.98 rz 89.74 deg; joints [-17.001, -74.603, 97.108, 11.751, 42.16, -23.892]
  MoveL 914 to (-1700.62, 22.36, -47.24) mm, rotated rx 0 ry 63.12 rz 89.75 deg; joints [-17.112, -74.586, 97.115, 11.733, 42.282, -23.984]
  MoveL 915 to (-1704.86, 23.61, -49.69) mm, rotated rx 0 ry 63.29 rz 89.76 deg; joints [-17.218, -74.578, 97.139, 11.693, 42.422, -24.057]
  MoveL 916 to (-1708.8, 25.04, -52.51) mm, rotated rx 0 ry 63.48 rz 89.76 deg; joints [-17.319, -74.58, 97.179, 11.631, 42.58, -24.112]
  MoveL 917 to (-1712.4, 26.63, -55.68) mm, rotated rx 0 ry 63.7 rz 89.78 deg; joints [-17.413, -74.591, 97.235, 11.549, 42.751, -24.147]
  MoveL 918 to (-1718.48, 30.19, -62.91) mm, rotated rx 0 ry 64.21 rz 89.81 deg; joints [-17.579, -74.643, 97.395, 11.327, 43.123, -24.162]
  MoveL 919 to (-1722.91, 34.1, -71.09) mm, rotated rx 0 ry 64.77 rz 89.85 deg; joints [-17.709, -74.732, 97.613, 11.04, 43.514, -24.108]
  MoveL 920 to (-1725.61, 38.21, -79.92) mm, rotated rx 0 ry 65.35 rz 89.91 deg; joints [-17.802, -74.857, 97.884, 10.705, 43.9, -23.993]
  MoveL 921 to (-1726.52, 42.36, -89.09) mm, rotated rx 0 ry 65.94 rz 89.98 deg; joints [-17.855, -75.015, 98.201, 10.341, 44.26, -23.829]
  MoveL 922 to (-1726.52, 42.36, -89.09) mm, rotated rx 0 ry 65.94 rz 89.98 deg; joints [-17.855, -75.015, 98.201, 10.341, 44.26, -23.829]
  MoveL 923 to (-1726.52, 68.06, -148.79) mm, rotated rx 0 ry 64.87 rz 88.95 deg; joints [-18.505, -76.852, 101.818, 12.984, 42.069, -26.164]
  MoveL 924 to (-1726.52, 75.02, -162.53) mm, rotated rx 0 ry 60.92 rz 87.34 deg; joints [-19.019, -77.722, 103.779, 18.484, 38.337, -30.284]
  MoveL 925 to (-1726.52, 82.57, -174.64) mm, rotated rx 0 ry 54.96 rz 84.8 deg; joints [-19.709, -78.61, 106.24, 28.587, 33.402, -38.084]
  MoveL 926 to (-1726.52, 91.33, -185.47) mm, rotated rx 0 ry 47.27 rz 81.01 deg; joints [-20.535, -79.268, 109.077, 45.999, 28.708, -51.961]
  MoveL 927 to (-1726.52, 96.32, -190.41) mm, rotated rx 0 ry 43.06 rz 78.54 deg; joints [-20.959, -79.412, 110.529, 57.688, 27.33, -61.325]
  MoveL 928 to (-1726.52, 101.81, -195.05) mm, rotated rx 0 ry 38.82 rz 75.65 deg; joints [-21.365, -79.397, 111.935, 70.437, 27.047, -71.333]
  MoveL 929 to (-1726.52, 107.85, -199.39) mm, rotated rx 0 ry 34.8 rz 72.34 deg; joints [-21.732, -79.219, 113.226, 82.639, 27.952, -80.38]
  MoveL 930 to (-1726.52, 114.5, -203.45) mm, rotated rx 0 ry 31.13 rz 68.6 deg; joints [-22.052, -78.894, 114.376, 93.173, 29.799, -87.349]
  MoveL 931 to (-1726.52, 121.82, -207.24) mm, rotated rx 0 ry 27.89 rz 64.48 deg; joints [-22.322, -78.454, 115.378, 101.665, 32.218, -91.898]
  MoveL 932 to (-1726.52, 129.87, -210.78) mm, rotated rx 0 ry 25.12 rz 60.04 deg; joints [-22.544, -77.929, 116.238, 108.284, 34.877, -94.268]
  MoveL 933 to (-1726.52, 138.73, -214.1) mm, rotated rx 0 ry 22.82 rz 55.39 deg; joints [-22.724, -77.348, 116.972, 113.398, 37.545, -94.934]
  MoveL 934 to (-1726.52, 148.47, -217.22) mm, rotated rx 0 ry 20.96 rz 50.65 deg; joints [-22.868, -76.729, 117.601, 117.381, 40.093, -94.391]
  MoveL 935 to (-1726.52, 159.21, -220.17) mm, rotated rx 0 ry 19.47 rz 45.94 deg; joints [-22.984, -76.082, 118.147, 120.537, 42.466, -93.065]
  MoveL 936 to (-1726.52, 171.05, -222.96) mm, rotated rx 0 ry 18.3 rz 41.41 deg; joints [-23.077, -75.413, 118.626, 123.077, 44.643, -91.305]
  MoveL 937 to (-1726.52, 184.08, -225.6) mm, rotated rx 0 ry 17.39 rz 37.15 deg; joints [-23.152, -74.721, 119.052, 125.157, 46.625, -89.383]
  MoveL 938 to (-1726.52, 198.36, -228.12) mm, rotated rx 0 ry 16.7 rz 33.25 deg; joints [-23.213, -74.005, 119.435, 126.893, 48.429, -87.496]
  MoveL 939 to (-1726.52, 214.01, -230.53) mm, rotated rx 0 ry 16.16 rz 29.76 deg; joints [-23.263, -73.258, 119.785, 128.369, 50.081, -85.776]
  MoveL 940 to (-1726.52, 231.09, -232.83) mm, rotated rx 0 ry 15.75 rz 26.69 deg; joints [-23.305, -72.474, 120.107, 129.648, 51.606, -84.3]
  MoveL 941 to (-1726.52, 249.69, -235.05) mm, rotated rx 0 ry 15.43 rz 24.02 deg; joints [-23.341, -71.644, 120.406, 130.776, 53.029, -83.107]
  MoveL 942 to (-1726.52, 269.91, -237.19) mm, rotated rx 0 ry 15.18 rz 21.73 deg; joints [-23.371, -70.761, 120.683, 131.789, 54.376, -82.206]
  MoveL 943 to (-1726.52, 291.83, -239.28) mm, rotated rx 0 ry 14.97 rz 19.79 deg; joints [-23.397, -69.816, 120.939, 132.713, 55.667, -81.591]
  MoveL 944 to (-1726.52, 315.53, -241.33) mm, rotated rx 0 ry 14.81 rz 18.16 deg; joints [-23.421, -68.8, 121.174, 133.567, 56.924, -81.248]
  MoveL 945 to (-1726.52, 315.53, -241.33) mm, rotated rx 0 ry 14.81 rz 18.16 deg; joints [-23.421, -68.8, 121.174, 133.567, 56.924, -81.248]
  MoveL 946 to (-1727.34, 327.53, -242.09) mm, rotated rx 0 ry 14.75 rz 17.47 deg; joints [-23.451, -68.271, 121.253, 133.925, 57.521, -81.15]
  MoveL 947 to (-1729.71, 339.3, -242.41) mm, rotated rx 0 ry 14.7 rz 16.87 deg; joints [-23.516, -67.723, 121.274, 134.193, 58.089, -81.065]
  MoveL 948 to (-1733.53, 350.65, -242.3) mm, rotated rx 0 ry 14.67 rz 16.36 deg; joints [-23.614, -67.167, 121.239, 134.375, 58.619, -80.985]
  MoveL 949 to (-1738.73, 361.39, -241.77) mm, rotated rx 0 ry 14.66 rz 15.92 deg; joints [-23.744, -66.613, 121.149, 134.473, 59.105, -80.903]
  MoveL 950 to (-1745.27, 371.22, -240.82) mm, rotated rx 0 ry 14.66 rz 15.55 deg; joints [-23.904, -66.075, 121.005, 134.486, 59.539, -80.81]
  MoveL 951 to (-1753.11, 379.89, -239.45) mm, rotated rx 0 ry 14.68 rz 15.26 deg; joints [-24.092, -65.565, 120.808, 134.412, 59.911, -80.693]
  MoveL 952 to (-1757.5, 383.65, -238.59) mm, rotated rx 0 ry 14.69 rz 15.14 deg; joints [-24.197, -65.326, 120.689, 134.341, 60.071, -80.622]
  MoveL 953 to (-1762.2, 386.97, -237.63) mm, rotated rx 0 ry 14.71 rz 15.03 deg; joints [-24.307, -65.101, 120.557, 134.248, 60.209, -80.54]
  MoveL 954 to (-1767.16, 389.75, -236.56) mm, rotated rx 0 ry 14.73 rz 14.95 deg; joints [-24.424, -64.895, 120.413, 134.131, 60.325, -80.446]
  MoveL 955 to (-1772.37, 391.94, -235.38) mm, rotated rx 0 ry 14.76 rz 14.88 deg; joints [-24.545, -64.709, 120.257, 133.991, 60.416, -80.34]
  MoveL 956 to (-1777.75, 393.43, -234.11) mm, rotated rx 0 ry 14.79 rz 14.84 deg; joints [-24.669, -64.55, 120.092, 133.828, 60.478, -80.22]
  MoveL 957 to (-1783.24, 394.16, -232.76) mm, rotated rx 0 ry 14.82 rz 14.81 deg; joints [-24.795, -64.421, 119.918, 133.644, 60.51, -80.086]
  MoveL 958 to (-1788.73, 394.07, -231.35) mm, rotated rx 0 ry 14.85 rz 14.81 deg; joints [-24.919, -64.326, 119.74, 133.441, 60.51, -79.94]
  MoveL 959 to (-1794.09, 393.15, -229.91) mm, rotated rx 0 ry 14.89 rz 14.83 deg; joints [-25.04, -64.268, 119.561, 133.223, 60.478, -79.784]
  MoveL 960 to (-1799.24, 391.38, -228.47) mm, rotated rx 0 ry 14.93 rz 14.88 deg; joints [-25.155, -64.249, 119.384, 132.994, 60.413, -79.622]
  MoveL 961 to (-1804.01, 388.86, -227.06) mm, rotated rx 0 ry 14.96 rz 14.94 deg; joints [-25.261, -64.267, 119.214, 132.759, 60.32, -79.458]
  MoveL 962 to (-1808.37, 385.65, -225.71) mm, rotated rx 0 ry 15 rz 15.03 deg; joints [-25.356, -64.319, 119.054, 132.523, 60.201, -79.296]
  MoveL 963 to (-1812.27, 381.86, -224.44) mm, rotated rx 0 ry 15.04 rz 15.14 deg; joints [-25.44, -64.404, 118.905, 132.288, 60.058, -79.139]
  MoveL 964 to (-1815.66, 377.6, -223.25) mm, rotated rx 0 ry 15.07 rz 15.27 deg; joints [-25.513, -64.516, 118.768, 132.059, 59.898, -78.992]
  MoveL 965 to (-1818.56, 372.97, -222.17) mm, rotated rx 0 ry 15.11 rz 15.41 deg; joints [-25.574, -64.652, 118.645, 131.836, 59.721, -78.856]
  MoveL 966 to (-1820.98, 368.04, -221.19) mm, rotated rx 0 ry 15.14 rz 15.57 deg; joints [-25.624, -64.808, 118.535, 131.62, 59.531, -78.734]
  MoveL 967 to (-1822.96, 362.79, -220.29) mm, rotated rx 0 ry 15.17 rz 15.75 deg; joints [-25.664, -64.984, 118.436, 131.41, 59.327, -78.624]
  MoveL 968 to (-1824.51, 357.25, -219.47) mm, rotated rx 0 ry 15.21 rz 15.95 deg; joints [-25.694, -65.18, 118.348, 131.203, 59.108, -78.529]
  MoveL 969 to (-1825.62, 351.45, -218.74) mm, rotated rx 0 ry 15.24 rz 16.17 deg; joints [-25.714, -65.394, 118.271, 131.001, 58.876, -78.451]
  MoveL 970 to (-1826.52, 339.29, -217.57) mm, rotated rx 0 ry 15.3 rz 16.67 deg; joints [-25.724, -65.87, 118.151, 130.616, 58.373, -78.353]
  MoveL 971 to (-1826.52, 339.29, -217.57) mm, rotated rx 0 ry 15.3 rz 16.67 deg; joints [-25.724, -65.87, 118.151, 130.616, 58.373, -78.353]
  MoveL 972 to (-1826.52, 316.68, -215.73) mm, rotated rx 0 ry 15.42 rz 17.78 deg; joints [-25.703, -66.784, 117.964, 129.902, 57.386, -78.334]
  MoveL 973 to (-1826.52, 295.48, -213.88) mm, rotated rx 0 ry 15.55 rz 19.09 deg; joints [-25.681, -67.64, 117.758, 129.147, 56.387, -78.488]
  MoveL 974 to (-1826.52, 275.63, -211.99) mm, rotated rx 0 ry 15.72 rz 20.6 deg; joints [-25.657, -68.444, 117.537, 128.341, 55.367, -78.828]
  MoveL 975 to (-1826.52, 257.08, -210.07) mm, rotated rx 0 ry 15.91 rz 22.34 deg; joints [-25.631, -69.2, 117.301, 127.473, 54.313, -79.363]
  MoveL 976 to (-1826.52, 239.76, -208.11) mm, rotated rx 0 ry 16.15 rz 24.34 deg; joints [-25.602, -69.914, 117.049, 126.528, 53.215, -80.099]
  MoveL 977 to (-1826.52, 223.63, -206.08) mm, rotated rx 0 ry 16.44 rz 26.61 deg; joints [-25.568, -70.591, 116.781, 125.487, 52.059, -81.037]
  MoveL 978 to (-1826.52, 208.63, -203.99) mm, rotated rx 0 ry 16.8 rz 29.17 deg; joints [-25.53, -71.236, 116.495, 124.328, 50.832, -82.168]
  MoveL 979 to (-1826.52, 194.7, -201.83) mm, rotated rx 0 ry 17.24 rz 32.04 deg; joints [-25.485, -71.854, 116.189, 123.02, 49.519, -83.469]
  MoveL 980 to (-1826.52, 181.79, -199.57) mm, rotated rx 0 ry 17.8 rz 35.19 deg; joints [-25.433, -72.448, 115.859, 121.525, 48.105, -84.895]
  MoveL 981 to (-1826.52, 169.85, -197.23) mm, rotated rx 0 ry 18.49 rz 38.62 deg; joints [-25.372, -73.023, 115.5, 119.796, 46.578, -86.381]
  MoveL 982 to (-1826.52, 158.82, -194.78) mm, rotated rx 0 ry 19.36 rz 42.29 deg; joints [-25.299, -73.58, 115.107, 117.77, 44.928, -87.827]
  MoveL 983 to (-1826.52, 148.64, -192.22) mm, rotated rx 0 ry 20.43 rz 46.14 deg; joints [-25.211, -74.12, 114.671, 115.369, 43.149, -89.099]
  MoveL 984 to (-1826.52, 139.27, -189.53) mm, rotated rx 0 ry 21.73 rz 50.12 deg; joints [-25.106, -74.644, 114.185, 112.493, 41.247, -90.026]
  MoveL 985 to (-1826.52, 130.64, -186.71) mm, rotated rx 0 ry 23.31 rz 54.12 deg; joints [-24.978, -75.145, 113.639, 109.037, 39.242, -90.416]
  MoveL 986 to (-1826.52, 122.68, -183.74) mm, rotated rx 0 ry 25.18 rz 58.08 deg; joints [-24.825, -75.62, 113.022, 104.836, 37.174, -90.029]
  MoveL 987 to (-1826.52, 115.33, -180.6) mm, rotated rx 0 ry 27.37 rz 61.93 deg; joints [-24.642, -76.057, 112.32, 99.712, 35.11, -88.611]
  MoveL 988 to (-1826.52, 108.55, -177.29) mm, rotated rx 0 ry 29.89 rz 65.58 deg; joints [-24.424, -76.443, 111.525, 93.5, 33.167, -85.926]
  MoveL 989 to (-1826.52, 102.29, -173.78) mm, rotated rx 0 ry 32.72 rz 68.99 deg; joints [-24.171, -76.76, 110.631, 86.105, 31.499, -81.82]
  MoveL 990 to (-1826.52, 91.17, -166.15) mm, rotated rx 0 ry 39.14 rz 74.95 deg; joints [-23.559, -77.122, 108.558, 68.259, 29.704, -69.714]
  MoveL 991 to (-1826.52, 81.67, -157.63) mm, rotated rx 0 ry 46.02 rz 79.69 deg; joints [-22.847, -77.058, 106.214, 49.563, 30.678, -55.569]
  MoveL 992 to (-1826.52, 73.51, -148.24) mm, rotated rx 0 ry 52.49 rz 83.27 deg; joints [-22.125, -76.62, 103.847, 34.528, 33.819, -43.944]
  MoveL 993 to (-1826.52, 66.38, -137.99) mm, rotated rx 0 ry 57.86 rz 85.86 deg; joints [-21.48, -75.971, 101.697, 24.364, 37.591, -36.207]
  MoveL 994 to (-1826.52, 59.93, -126.86) mm, rotated rx 0 ry 61.82 rz 87.68 deg; joints [-20.958, -75.279, 99.892, 18.006, 40.875, -31.488]
  MoveL 995 to (-1826.52, 53.77, -114.64) mm, rotated rx 0 ry 64.4 rz 88.9 deg; joints [-20.563, -74.643, 98.437, 14.193, 43.245, -28.704]
  MoveL 996 to (-1826.52, 47.58, -101.27) mm, rotated rx 0 ry 65.73 rz 89.67 deg; joints [-20.279, -74.106, 97.294, 12.11, 44.632, -27.176]
  MoveL 997 to (-1826.52, 47.58, -101.27) mm, rotated rx 0 ry 65.73 rz 89.67 deg; joints [-20.279, -74.106, 97.294, 12.11, 44.632, -27.176]
  MoveL 998 to (-1827.41, 43.47, -92.07) mm, rotated rx 0 ry 66.01 rz 89.96 deg; joints [-20.169, -73.807, 96.688, 11.471, 45.039, -26.698]
  MoveL 999 to (-1830.08, 39.49, -83.16) mm, rotated rx 0 ry 65.93 rz 90.13 deg; joints [-20.137, -73.542, 96.175, 11.267, 45.139, -26.557]
  MoveL 1000 to (-1834.45, 35.76, -74.87) mm, rotated rx 0 ry 65.65 rz 90.21 deg; joints [-20.17, -73.301, 95.73, 11.332, 45.056, -26.638]
  MoveL 1001 to (-1840.45, 32.37, -67.5) mm, rotated rx 0 ry 65.18 rz 90.2 deg; joints [-20.267, -73.089, 95.36, 11.657, 44.815, -26.931]
  MoveL 1002 to (-1844.01, 30.85, -64.27) mm, rotated rx 0 ry 64.93 rz 90.18 deg; joints [-20.334, -72.99, 95.193, 11.86, 44.68, -27.119]
  MoveL 1003 to (-1847.9, 29.48, -61.38) mm, rotated rx 0 ry 64.71 rz 90.17 deg; joints [-20.41, -72.892, 95.032, 12.048, 44.564, -27.306]
  MoveL 1004 to (-1852.1, 28.28, -58.86) mm, rotated rx 0 ry 64.52 rz 90.16 deg; joints [-20.493, -72.795, 94.875, 12.217, 44.471, -27.489]
  MoveL 1005 to (-1856.57, 27.26, -56.75) mm, rotated rx 0 ry 64.36 rz 90.16 deg; joints [-20.582, -72.701, 94.726, 12.365, 44.403, -27.665]
  MoveL 1006 to (-1861.25, 26.44, -55.07) mm, rotated rx 0 ry 64.24 rz 90.15 deg; joints [-20.678, -72.61, 94.585, 12.489, 44.363, -27.832]
  MoveL 1007 to (-1866.12, 25.83, -53.85) mm, rotated rx 0 ry 64.16 rz 90.16 deg; joints [-20.778, -72.522, 94.453, 12.585, 44.354, -27.985]
  MoveL 1008 to (-1871.1, 25.45, -53.1) mm, rotated rx 0 ry 64.12 rz 90.17 deg; joints [-20.882, -72.438, 94.331, 12.65, 44.377, -28.123]
  MoveL 1009 to (-1876.14, 25.31, -52.83) mm, rotated rx 0 ry 64.13 rz 90.18 deg; joints [-20.988, -72.36, 94.22, 12.682, 44.434, -28.241]
  MoveL 1010 to (-1881.19, 25.39, -53.05) mm, rotated rx 0 ry 64.18 rz 90.19 deg; joints [-21.096, -72.287, 94.121, 12.68, 44.525, -28.339]
  MoveL 1011 to (-1886.17, 25.72, -53.75) mm, rotated rx 0 ry 64.2 rz 90.17 deg; joints [-21.213, -72.232, 94.061, 12.761, 44.578, -28.49]
  MoveL 1012 to (-1891.05, 26.27, -54.92) mm, rotated rx 0 ry 64.22 rz 90.13 deg; joints [-21.334, -72.189, 94.025, 12.858, 44.632, -28.652]
  MoveL 1013 to (-1895.77, 27.04, -56.54) mm, rotated rx 0 ry 64.25 rz 90.07 deg; joints [-21.456, -72.158, 94.016, 12.971, 44.685, -28.822]
  MoveL 1014 to (-1900.27, 28.03, -58.59) mm, rotated rx 0 ry 64.27 rz 90 deg; joints [-21.58, -72.142, 94.035, 13.112, 44.726, -29.009]
  MoveL 1015 to (-1904.52, 29.21, -61.04) mm, rotated rx 0 ry 64.27 rz 89.91 deg; joints [-21.705, -72.141, 94.087, 13.296, 44.743, -29.22]
  MoveL 1016 to (-1912.09, 32.13, -67.02) mm, rotated rx 0 ry 64.15 rz 89.64 deg; joints [-21.964, -72.195, 94.305, 13.864, 44.65, -29.766]
  MoveL 1017 to (-1918.24, 35.69, -74.18) mm, rotated rx 0 ry 63.72 rz 89.21 deg; joints [-22.238, -72.336, 94.707, 14.852, 44.283, -30.577]
  MoveL 1018 to (-1922.78, 39.8, -82.2) mm, rotated rx 0 ry 62.83 rz 88.58 deg; joints [-22.536, -72.573, 95.328, 16.483, 43.515, -31.807]
  MoveL 1019 to (-1925.57, 44.41, -90.73) mm, rotated rx 0 ry 61.31 rz 87.69 deg; joints [-22.867, -72.911, 96.199, 19.018, 42.25, -33.65]
  MoveL 1020 to (-1926.52, 49.42, -99.42) mm, rotated rx 0 ry 59.1 rz 86.5 deg; joints [-23.23, -73.331, 97.321, 22.708, 40.491, -36.308]
  MoveL 1021 to (-1926.52, 49.42, -99.42) mm, rotated rx 0 ry 59.1 rz 86.5 deg; joints [-23.23, -73.331, 97.321, 22.708, 40.491, -36.308]
  MoveL 1022 to (-1926.52, 55.74, -109.28) mm, rotated rx 0 ry 55.56 rz 84.65 deg; joints [-23.719, -73.862, 98.915, 28.988, 37.933, -40.878]
  MoveL 1023 to (-1926.52, 62.54, -118.37) mm, rotated rx 0 ry 51.07 rz 82.2 deg; joints [-24.286, -74.333, 100.724, 37.936, 35.238, -47.495]
  MoveL 1024 to (-1926.52, 70.03, -126.73) mm, rotated rx 0 ry 45.86 rz 79.04 deg; joints [-24.897, -74.648, 102.657, 49.79, 33.085, -56.301]
  MoveL 1025 to (-1926.52, 78.45, -134.41) mm, rotated rx 0 ry 40.35 rz 75.09 deg; joints [-25.499, -74.721, 104.579, 63.752, 32.239, -66.414]
  MoveL 1026 to (-1926.52, 87.97, -141.42) mm, rotated rx 0 ry 35.02 rz 70.29 deg; joints [-26.042, -74.517, 106.352, 77.759, 33.08, -75.745]
  MoveL 1027 to (-1926.52, 98.79, -147.8) mm, rotated rx 0 ry 30.27 rz 64.69 deg; joints [-26.493, -74.063, 107.89, 89.822, 35.319, -82.35]
  MoveL 1028 to (-1926.52, 111.14, -153.63) mm, rotated rx 0 ry 26.33 rz 58.44 deg; joints [-26.845, -73.424, 109.171, 99.201, 38.305, -85.651]
  MoveL 1029 to (-1926.52, 125.23, -158.94) mm, rotated rx 0 ry 23.27 rz 51.83 deg; joints [-27.109, -72.669, 110.218, 106.168, 41.46, -86.217]
  MoveL 1030 to (-1926.52, 133.02, -161.43) mm, rotated rx 0 ry 22.04 rz 48.5 deg; joints [-27.214, -72.262, 110.669, 108.936, 42.991, -85.776]
  MoveL 1031 to (-1926.52, 141.35, -163.83) mm, rotated rx 0 ry 20.99 rz 45.22 deg; joints [-27.304, -71.84, 111.079, 111.326, 44.459, -85.012]
  MoveL 1032 to (-1926.52, 150.26, -166.13) mm, rotated rx 0 ry 20.1 rz 42.03 deg; joints [-27.382, -71.405, 111.456, 113.4, 45.854, -84.035]
  MoveL 1033 to (-1926.52, 159.79, -168.34) mm, rotated rx 0 ry 19.35 rz 38.97 deg; joints [-27.449, -70.958, 111.802, 115.209, 47.168, -82.936]
  MoveL 1034 to (-1926.52, 169.96, -170.48) mm, rotated rx 0 ry 18.72 rz 36.07 deg; joints [-27.506, -70.499, 112.123, 116.797, 48.404, -81.793]
  MoveL 1035 to (-1926.52, 180.81, -172.54) mm, rotated rx 0 ry 18.2 rz 33.35 deg; joints [-27.557, -70.026, 112.422, 118.202, 49.563, -80.667]
  MoveL 1036 to (-1926.52, 192.37, -174.53) mm, rotated rx 0 ry 17.76 rz 30.84 deg; joints [-27.6, -69.537, 112.703, 119.454, 50.652, -79.603]
  MoveL 1037 to (-1926.52, 204.67, -176.45) mm, rotated rx 0 ry 17.4 rz 28.53 deg; joints [-27.639, -69.032, 112.967, 120.578, 51.677, -78.634]
  MoveL 1038 to (-1926.52, 217.75, -178.33) mm, rotated rx 0 ry 17.1 rz 26.43 deg; joints [-27.673, -68.507, 113.217, 121.597, 52.646, -77.782]
  MoveL 1039 to (-1926.52, 231.64, -180.15) mm, rotated rx 0 ry 16.84 rz 24.53 deg; joints [-27.704, -67.959, 113.453, 122.527, 53.566, -77.059]
  MoveL 1040 to (-1926.52, 246.38, -181.93) mm, rotated rx 0 ry 16.63 rz 22.83 deg; joints [-27.732, -67.387, 113.678, 123.382, 54.446, -76.472]
  MoveL 1041 to (-1926.52, 261.99, -183.66) mm, rotated rx 0 ry 16.45 rz 21.3 deg; joints [-27.757, -66.787, 113.892, 124.176, 55.291, -76.021]
  MoveL 1042 to (-1926.52, 278.5, -185.37) mm, rotated rx 0 ry 16.29 rz 19.94 deg; joints [-27.781, -66.156, 114.094, 124.917, 56.109, -75.706]
  MoveL 1043 to (-1926.52, 295.96, -187.05) mm, rotated rx 0 ry 16.15 rz 18.74 deg; joints [-27.802, -65.491, 114.285, 125.615, 56.907, -75.522]
  MoveL 1044 to (-1926.52, 314.39, -188.71) mm, rotated rx 0 ry 16.04 rz 17.68 deg; joints [-27.823, -64.79, 114.464, 126.275, 57.689, -75.463]
  MoveL 1045 to (-1926.52, 333.82, -190.36) mm, rotated rx 0 ry 15.93 rz 16.75 deg; joints [-27.842, -64.048, 114.63, 126.905, 58.462, -75.522]
  MoveL 1046 to (-1926.52, 333.82, -190.36) mm, rotated rx 0 ry 15.93 rz 16.75 deg; joints [-27.842, -64.048, 114.63, 126.905, 58.462, -75.522]
  MoveL 1047 to (-1927.36, 345.98, -191.11) mm, rotated rx 0 ry 15.88 rz 16.25 deg; joints [-27.87, -63.566, 114.693, 127.24, 58.925, -75.587]
  MoveL 1048 to (-1929.82, 358.04, -191.39) mm, rotated rx 0 ry 15.84 rz 15.8 deg; joints [-27.931, -63.053, 114.69, 127.497, 59.373, -75.642]
  MoveL 1049 to (-1933.77, 369.65, -191.2) mm, rotated rx 0 ry 15.82 rz 15.42 deg; joints [-28.021, -62.528, 114.622, 127.673, 59.793, -75.68]
  MoveL 1050 to (-1939.1, 380.53, -190.55) mm, rotated rx 0 ry 15.82 rz 15.09 deg; joints [-28.139, -62.002, 114.493, 127.77, 60.177, -75.693]
  MoveL 1051 to (-1945.76, 390.48, -189.45) mm, rotated rx 0 ry 15.82 rz 14.82 deg; joints [-28.281, -61.486, 114.304, 127.787, 60.52, -75.674]
  MoveL 1052 to (-1953.69, 399.19, -187.9) mm, rotated rx 0 ry 15.84 rz 14.6 deg; joints [-28.448, -60.994, 114.058, 127.724, 60.813, -75.613]
  MoveL 1053 to (-1958.12, 402.97, -186.96) mm, rotated rx 0 ry 15.86 rz 14.51 deg; joints [-28.539, -60.761, 113.914, 127.662, 60.938, -75.563]
  MoveL 1054 to (-1962.82, 406.29, -185.9) mm, rotated rx 0 ry 15.87 rz 14.43 deg; joints [-28.636, -60.541, 113.756, 127.578, 61.046, -75.499]
  MoveL 1055 to (-1967.77, 409.07, -184.73) mm, rotated rx 0 ry 15.9 rz 14.37 deg; joints [-28.737, -60.336, 113.585, 127.473, 61.137, -75.418]
  MoveL 1056 to (-1972.94, 411.25, -183.46) mm, rotated rx 0 ry 15.92 rz 14.32 deg; joints [-28.841, -60.15, 113.403, 127.347, 61.208, -75.321]
  MoveL 1057 to (-1978.28, 412.76, -182.09) mm, rotated rx 0 ry 15.95 rz 14.29 deg; joints [-28.948, -59.986, 113.211, 127.2, 61.257, -75.205]
  MoveL 1058 to (-1983.69, 413.52, -180.64) mm, rotated rx 0 ry 15.98 rz 14.27 deg; joints [-29.055, -59.849, 113.012, 127.034, 61.283, -75.073]
  MoveL 1059 to (-1989.08, 413.49, -179.14) mm, rotated rx 0 ry 16.01 rz 14.27 deg; joints [-29.161, -59.743, 112.809, 126.851, 61.285, -74.925]
  MoveL 1060 to (-1994.38, 412.63, -177.61) mm, rotated rx 0 ry 16.04 rz 14.29 deg; joints [-29.263, -59.669, 112.606, 126.653, 61.261, -74.763]
  MoveL 1061 to (-1999.41, 410.96, -176.08) mm, rotated rx 0 ry 16.08 rz 14.32 deg; joints [-29.36, -59.63, 112.409, 126.446, 61.214, -74.592]
  MoveL 1062 to (-2004.11, 408.56, -174.6) mm, rotated rx 0 ry 16.12 rz 14.37 deg; joints [-29.449, -59.625, 112.22, 126.233, 61.145, -74.415]
  MoveL 1063 to (-2008.41, 405.47, -173.17) mm, rotated rx 0 ry 16.15 rz 14.44 deg; joints [-29.53, -59.652, 112.042, 126.017, 61.055, -74.236]
  MoveL 1064 to (-2012.23, 401.84, -171.83) mm, rotated rx 0 ry 16.18 rz 14.52 deg; joints [-29.601, -59.709, 111.879, 125.804, 60.948, -74.06]
  MoveL 1065 to (-2015.57, 397.75, -170.6) mm, rotated rx 0 ry 16.22 rz 14.62 deg; joints [-29.661, -59.792, 111.732, 125.596, 60.828, -73.891]
  MoveL 1066 to (-2018.44, 393.27, -169.46) mm, rotated rx 0 ry 16.25 rz 14.72 deg; joints [-29.713, -59.897, 111.599, 125.392, 60.695, -73.729]
  MoveL 1067 to (-2020.88, 388.4, -168.41) mm, rotated rx 0 ry 16.28 rz 14.85 deg; joints [-29.755, -60.026, 111.48, 125.191, 60.549, -73.575]
  MoveL 1068 to (-2022.9, 383.17, -167.44) mm, rotated rx 0 ry 16.31 rz 14.98 deg; joints [-29.789, -60.175, 111.373, 124.994, 60.391, -73.429]
  MoveL 1069 to (-2024.48, 377.61, -166.57) mm, rotated rx 0 ry 16.34 rz 15.14 deg; joints [-29.815, -60.345, 111.28, 124.799, 60.221, -73.293]
  MoveL 1070 to (-2025.62, 371.78, -165.8) mm, rotated rx 0 ry 16.37 rz 15.3 deg; joints [-29.831, -60.534, 111.201, 124.61, 60.04, -73.17]
  MoveL 1071 to (-2026.52, 359.59, -164.59) mm, rotated rx 0 ry 16.42 rz 15.68 deg; joints [-29.838, -60.958, 111.087, 124.252, 59.652, -72.972]
  MoveL 1072 to (-2026.52, 359.59, -164.59) mm, rotated rx 0 ry 16.42 rz 15.68 deg; joints [-29.838, -60.958, 111.087, 124.252, 59.652, -72.972]
  MoveL 1073 to (-2026.52, 342.79, -163.22) mm, rotated rx 0 ry 16.49 rz 16.28 deg; joints [-29.822, -61.567, 110.966, 123.772, 59.095, -72.777]
  MoveL 1074 to (-2026.52, 326.64, -161.85) mm, rotated rx 0 ry 16.57 rz 16.94 deg; joints [-29.805, -62.149, 110.836, 123.275, 58.536, -72.646]
  MoveL 1075 to (-2026.52, 311.13, -160.48) mm, rotated rx 0 ry 16.66 rz 17.68 deg; joints [-29.788, -62.707, 110.698, 122.76, 57.973, -72.582]
  MoveL 1076 to (-2026.52, 296.24, -159.09) mm, rotated rx 0 ry 16.75 rz 18.49 deg; joints [-29.771, -63.24, 110.552, 122.224, 57.403, -72.588]
  MoveL 1077 to (-2026.52, 281.97, -157.69) mm, rotated rx 0 ry 16.86 rz 19.39 deg; joints [-29.752, -63.752, 110.398, 121.664, 56.824, -72.668]
  MoveL 1078 to (-2026.52, 268.29, -156.28) mm, rotated rx 0 ry 16.97 rz 20.38 deg; joints [-29.733, -64.242, 110.236, 121.078, 56.234, -72.823]
  MoveL 1079 to (-2026.52, 255.19, -154.85) mm, rotated rx 0 ry 17.11 rz 21.46 deg; joints [-29.713, -64.713, 110.068, 120.461, 55.629, -73.057]
  MoveL 1080 to (-2026.52, 242.64, -153.39) mm, rotated rx 0 ry 17.25 rz 22.65 deg; joints [-29.691, -65.166, 109.892, 119.809, 55.008, -73.369]
  MoveL 1081 to (-2026.52, 230.65, -151.91) mm, rotated rx 0 ry 17.42 rz 23.94 deg; joints [-29.668, -65.602, 109.709, 119.117, 54.367, -73.762]
  MoveL 1082 to (-2026.52, 219.18, -150.4) mm, rotated rx 0 ry 17.61 rz 25.35 deg; joints [-29.643, -66.023, 109.519, 118.38, 53.703, -74.235]
  MoveL 1083 to (-2026.52, 197.77, -147.29) mm, rotated rx 0 ry 18.08 rz 28.52 deg; joints [-29.586, -66.822, 109.114, 116.743, 52.294, -75.407]
  MoveL 1084 to (-2026.52, 178.29, -144.02) mm, rotated rx 0 ry 18.7 rz 32.18 deg; joints [-29.519, -67.574, 108.672, 114.833, 50.755, -76.84]
  MoveL 1085 to (-2026.52, 160.6, -140.59) mm, rotated rx 0 ry 19.52 rz 36.32 deg; joints [-29.436, -68.286, 108.186, 112.564, 49.065, -78.441]
  MoveL 1086 to (-2026.52, 144.58, -136.95) mm, rotated rx 0 ry 20.59 rz 40.9 deg; joints [-29.334, -68.964, 107.644, 109.828, 47.208, -80.046]
  MoveL 1087 to (-2026.52, 130.1, -133.09) mm, rotated rx 0 ry 21.99 rz 45.81 deg; joints [-29.206, -69.61, 107.033, 106.48, 45.186, -81.412]
  MoveL 1088 to (-2026.52, 117.03, -128.98) mm, rotated rx 0 ry 23.78 rz 50.91 deg; joints [-29.046, -70.221, 106.334, 102.346, 43.026, -82.212]
  MoveL 1089 to (-2026.52, 105.24, -124.59) mm, rotated rx 0 ry 26.03 rz 56.03 deg; joints [-28.843, -70.786, 105.527, 97.214, 40.799, -82.066]
  MoveL 1090 to (-2026.52, 94.57, -119.89) mm, rotated rx 0 ry 28.77 rz 61 deg; joints [-28.591, -71.289, 104.592, 90.87, 38.638, -80.583]
  MoveL 1091 to (-2026.52, 84.92, -114.84) mm, rotated rx 0 ry 31.99 rz 65.67 deg; joints [-28.282, -71.702, 103.518, 83.186, 36.748, -77.476]
  MoveL 1092 to (-2026.52, 76.17, -109.42) mm, rotated rx 0 ry 35.63 rz 69.91 deg; joints [-27.916, -71.997, 102.302, 74.255, 35.384, -72.72]
  MoveL 1093 to (-2026.52, 68.21, -103.61) mm, rotated rx 0 ry 39.54 rz 73.67 deg; joints [-27.499, -72.151, 100.965, 64.512, 34.773, -66.681]
  MoveL 1094 to (-2026.52, 68.21, -103.61) mm, rotated rx 0 ry 39.54 rz 73.67 deg; joints [-27.499, -72.151, 100.965, 64.512, 34.773, -66.681]
  MoveL 1095 to (-2026.77, 64.41, -100.42) mm, rotated rx 0 ry 41.57 rz 75.39 deg; joints [-27.278, -72.165, 100.243, 59.492, 34.794, -63.351]
  MoveL 1096 to (-2027.5, 60.84, -97.08) mm, rotated rx 0 ry 43.53 rz 76.92 deg; joints [-27.067, -72.129, 99.514, 54.745, 35.031, -60.111]
  MoveL 1097 to (-2028.71, 57.51, -93.63) mm, rotated rx 0 ry 45.35 rz 78.25 deg; joints [-26.873, -72.051, 98.797, 50.426, 35.432, -57.112]
  MoveL 1098 to (-2030.39, 54.42, -90.14) mm, rotated rx 0 ry 47 rz 79.4 deg; joints [-26.702, -71.938, 98.108, 46.617, 35.942, -54.442]
  MoveL 1099 to (-2032.52, 51.59, -86.66) mm, rotated rx 0 ry 48.45 rz 80.38 deg; joints [-26.559, -71.801, 97.461, 43.365, 36.502, -52.155]
  MoveL 1100 to (-2035.07, 49.02, -83.27) mm, rotated rx 0 ry 49.68 rz 81.18 deg; joints [-26.445, -71.65, 96.867, 40.678, 37.059, -50.268]
  MoveL 1101 to (-2041.34, 44.66, -76.92) mm, rotated rx 0 ry 51.5 rz 82.35 deg; joints [-26.312, -71.333, 95.857, 36.834, 38.037, -47.594]
  MoveL 1102 to (-2048.97, 41.35, -71.47) mm, rotated rx 0 ry 52.5 rz 83 deg; joints [-26.3, -71.029, 95.091, 34.732, 38.717, -46.173]
  MoveL 1103 to (-2057.68, 39.12, -67.2) mm, rotated rx 0 ry 52.81 rz 83.22 deg; joints [-26.401, -70.761, 94.567, 34.064, 39.064, -45.775]
  MoveL 1104 to (-2067.16, 38.05, -64.32) mm, rotated rx 0 ry 52.48 rz 83.04 deg; joints [-26.602, -70.538, 94.281, 34.655, 39.097, -46.262]
  MoveL 1105 to (-2077.03, 38.2, -62.92) mm, rotated rx 0 ry 51.56 rz 82.46 deg; joints [-26.896, -70.363, 94.237, 36.474, 38.849, -47.596]
  MoveL 1106 to (-2086.88, 39.65, -62.99) mm, rotated rx 0 ry 50.02 rz 81.45 deg; joints [-27.272, -70.229, 94.444, 39.6, 38.374, -49.815]
  MoveL 1107 to (-2096.32, 42.46, -64.43) mm, rotated rx 0 ry 47.87 rz 79.93 deg; joints [-27.721, -70.122, 94.905, 44.173, 37.768, -52.991]
  MoveL 1108 to (-2104.96, 46.65, -67.01) mm, rotated rx 0 ry 45.11 rz 77.87 deg; joints [-28.223, -70.014, 95.603, 50.256, 37.202, -57.116]
  MoveL 1109 to (-2112.46, 52.19, -70.47) mm, rotated rx 0 ry 41.88 rz 75.21 deg; joints [-28.749, -69.868, 96.492, 57.674, 36.914, -61.962]
  MoveL 1110 to (-2118.52, 58.96, -74.5) mm, rotated rx 0 ry 38.39 rz 71.97 deg; joints [-29.259, -69.655, 97.489, 65.858, 37.126, -66.98]
  MoveL 1111 to (-2122.95, 66.74, -78.83) mm, rotated rx 0 ry 34.97 rz 68.26 deg; joints [-29.713, -69.367, 98.505, 73.962, 37.911, -71.439]
  MoveL 1112 to (-2125.63, 75.25, -83.26) mm, rotated rx 0 ry 31.87 rz 64.28 deg; joints [-30.086, -69.025, 99.47, 81.259, 39.149, -74.806]
  MoveL 1113 to (-2126.52, 84.16, -87.66) mm, rotated rx 0 ry 29.24 rz 60.25 deg; joints [-30.366, -68.666, 100.351, 87.384, 40.613, -76.952]
  MoveL 1114 to (-2126.52, 84.16, -87.66) mm, rotated rx 0 ry 29.24 rz 60.25 deg; joints [-30.366, -68.666, 100.351, 87.384, 40.613, -76.952]
  MoveL 1115 to (-2126.52, 93.15, -91.75) mm, rotated rx 0 ry 27.09 rz 56.34 deg; joints [-30.575, -68.299, 101.115, 92.328, 42.123, -78.052]
  MoveL 1116 to (-2126.52, 102.86, -95.62) mm, rotated rx 0 ry 25.23 rz 52.32 deg; joints [-30.752, -67.888, 101.802, 96.601, 43.712, -78.381]
  MoveL 1117 to (-2126.52, 113.38, -99.29) mm, rotated rx 0 ry 23.65 rz 48.27 deg; joints [-30.901, -67.443, 102.42, 100.259, 45.308, -78.088]
  MoveL 1118 to (-2126.52, 124.76, -102.77) mm, rotated rx 0 ry 22.34 rz 44.28 deg; joints [-31.026, -66.971, 102.976, 103.381, 46.861, -77.343]
  MoveL 1119 to (-2126.52, 137.08, -106.09) mm, rotated rx 0 ry 21.25 rz 40.44 deg; joints [-31.13, -66.475, 103.48, 106.05, 48.34, -76.312]
  MoveL 1120 to (-2126.52, 150.41, -109.25) mm, rotated rx 0 ry 20.37 rz 36.81 deg; joints [-31.217, -65.957, 103.939, 108.341, 49.729, -75.144]
  MoveL 1121 to (-2126.52, 164.82, -112.26) mm, rotated rx 0 ry 19.66 rz 33.44 deg; joints [-31.291, -65.417, 104.361, 110.32, 51.024, -73.955]
  MoveL 1122 to (-2126.52, 180.37, -115.14) mm, rotated rx 0 ry 19.09 rz 30.37 deg; joints [-31.354, -64.851, 104.751, 112.044, 52.228, -72.834]
  MoveL 1123 to (-2126.52, 197.14, -117.91) mm, rotated rx 0 ry 18.63 rz 27.6 deg; joints [-31.408, -64.258, 105.114, 113.56, 53.348, -71.844]
  MoveL 1124 to (-2126.52, 215.19, -120.58) mm, rotated rx 0 ry 18.25 rz 25.14 deg; joints [-31.456, -63.632, 105.454, 114.906, 54.396, -71.021]
  MoveL 1125 to (-2126.52, 234.59, -123.16) mm, rotated rx 0 ry 17.95 rz 22.97 deg; joints [-31.498, -62.969, 105.772, 116.113, 55.381, -70.386]
  MoveL 1126 to (-2126.52, 255.41, -125.67) mm, rotated rx 0 ry 17.7 rz 21.08 deg; joints [-31.536, -62.265, 106.07, 117.209, 56.315, -69.947]
  MoveL 1127 to (-2126.52, 277.72, -128.11) mm, rotated rx 0 ry 17.49 rz 19.44 deg; joints [-31.57, -61.512, 106.348, 118.212, 57.209, -69.703]
  MoveL 1128 to (-2126.52, 301.6, -130.51) mm, rotated rx 0 ry 17.31 rz 18.04 deg; joints [-31.602, -60.707, 106.607, 119.141, 58.073, -69.648]
  MoveL 1129 to (-2126.52, 327.1, -132.88) mm, rotated rx 0 ry 17.17 rz 16.83 deg; joints [-31.632, -59.844, 106.844, 120.008, 58.917, -69.772]
  MoveL 1130 to (-2126.52, 354.3, -135.23) mm, rotated rx 0 ry 17.04 rz 15.82 deg; joints [-31.661, -58.917, 107.058, 120.824, 59.748, -70.064]
  MoveL 1131 to (-2126.52, 354.3, -135.23) mm, rotated rx 0 ry 17.04 rz 15.82 deg; joints [-31.661, -58.917, 107.058, 120.824, 59.748, -70.064]
  MoveL 1132 to (-2127.36, 366.45, -135.98) mm, rotated rx 0 ry 16.99 rz 15.43 deg; joints [-31.687, -58.481, 107.107, 121.132, 60.104, -70.212]
  MoveL 1133 to (-2129.78, 378.39, -136.23) mm, rotated rx 0 ry 16.96 rz 15.09 deg; joints [-31.741, -58.015, 107.082, 121.368, 60.447, -70.334]
  MoveL 1134 to (-2133.62, 389.84, -136) mm, rotated rx 0 ry 16.95 rz 14.79 deg; joints [-31.819, -57.534, 106.99, 121.533, 60.769, -70.425]
  MoveL 1135 to (-2138.81, 400.65, -135.3) mm, rotated rx 0 ry 16.94 rz 14.54 deg; joints [-31.919, -57.045, 106.832, 121.628, 61.067, -70.481]
  MoveL 1136 to (-2145.27, 410.58, -134.15) mm, rotated rx 0 ry 16.95 rz 14.32 deg; joints [-32.041, -56.558, 106.611, 121.653, 61.335, -70.494]
  MoveL 1137 to (-2153.03, 419.43, -132.52) mm, rotated rx 0 ry 16.97 rz 14.14 deg; joints [-32.183, -56.08, 106.327, 121.606, 61.569, -70.455]
  MoveL 1138 to (-2157.38, 423.33, -131.52) mm, rotated rx 0 ry 16.98 rz 14.07 deg; joints [-32.261, -55.85, 106.161, 121.554, 61.671, -70.413]
  MoveL 1139 to (-2162.01, 426.79, -130.41) mm, rotated rx 0 ry 17 rz 14 deg; joints [-32.344, -55.628, 105.981, 121.482, 61.761, -70.355]
  MoveL 1140 to (-2166.91, 429.75, -129.17) mm, rotated rx 0 ry 17.02 rz 13.95 deg; joints [-32.43, -55.419, 105.786, 121.391, 61.838, -70.278]
  MoveL 1141 to (-2172.03, 432.13, -127.82) mm, rotated rx 0 ry 17.05 rz 13.91 deg; joints [-32.519, -55.224, 105.579, 121.28, 61.9, -70.182]
  MoveL 1142 to (-2177.34, 433.86, -126.37) mm, rotated rx 0 ry 17.07 rz 13.88 deg; joints [-32.611, -55.047, 105.361, 121.149, 61.945, -70.067]
  MoveL 1143 to (-2182.77, 434.86, -124.82) mm, rotated rx 0 ry 17.1 rz 13.86 deg; joints [-32.704, -54.893, 105.133, 120.998, 61.973, -69.931]
  MoveL 1144 to (-2188.22, 435.07, -123.21) mm, rotated rx 0 ry 17.13 rz 13.86 deg; joints [-32.796, -54.765, 104.901, 120.831, 61.982, -69.777]
  MoveL 1145 to (-2193.57, 434.44, -121.56) mm, rotated rx 0 ry 17.17 rz 13.87 deg; joints [-32.885, -54.667, 104.669, 120.648, 61.971, -69.607]
  MoveL 1146 to (-2198.75, 432.97, -119.9) mm, rotated rx 0 ry 17.2 rz 13.9 deg; joints [-32.97, -54.602, 104.441, 120.454, 61.941, -69.423]
  MoveL 1147 to (-2203.57, 430.72, -118.28) mm, rotated rx 0 ry 17.24 rz 13.94 deg; joints [-33.049, -54.57, 104.224, 120.253, 61.892, -69.232]
  MoveL 1148 to (-2208, 427.74, -116.72) mm, rotated rx 0 ry 17.27 rz 13.99 deg; joints [-33.12, -54.57, 104.02, 120.049, 61.827, -69.037]
  MoveL 1149 to (-2211.97, 424.14, -115.25) mm, rotated rx 0 ry 17.31 rz 14.06 deg; joints [-33.182, -54.601, 103.833, 119.845, 61.747, -68.842]
  MoveL 1150 to (-2215.43, 420.05, -113.89) mm, rotated rx 0 ry 17.34 rz 14.14 deg; joints [-33.235, -54.659, 103.665, 119.646, 61.655, -68.654]
  MoveL 1151 to (-2218.38, 415.55, -112.65) mm, rotated rx 0 ry 17.37 rz 14.23 deg; joints [-33.28, -54.742, 103.516, 119.452, 61.552, -68.473]
  MoveL 1152 to (-2220.85, 410.72, -111.53) mm, rotated rx 0 ry 17.4 rz 14.32 deg; joints [-33.316, -54.846, 103.385, 119.264, 61.441, -68.3]
  MoveL 1153 to (-2222.88, 405.52, -110.51) mm, rotated rx 0 ry 17.43 rz 14.44 deg; joints [-33.344, -54.971, 103.27, 119.079, 61.321, -68.136]
  MoveL 1154 to (-2224.47, 399.99, -109.59) mm, rotated rx 0 ry 17.45 rz 14.56 deg; joints [-33.365, -55.116, 103.172, 118.898, 61.191, -67.981]
  MoveL 1155 to (-2225.61, 394.18, -108.78) mm, rotated rx 0 ry 17.48 rz 14.69 deg; joints [-33.378, -55.281, 103.09, 118.722, 61.052, -67.836]
  MoveL 1156 to (-2226.52, 382.01, -107.52) mm, rotated rx 0 ry 17.53 rz 15 deg; joints [-33.381, -55.659, 102.98, 118.389, 60.755, -67.589]
  MoveL 1157 to (-2226.52, 382.01, -107.52) mm, rotated rx 0 ry 17.53 rz 15 deg; joints [-33.381, -55.659, 102.98, 118.389, 60.755, -67.589]
  MoveL 1158 to (-2226.52, 359.4, -105.63) mm, rotated rx 0 ry 17.62 rz 15.64 deg; joints [-33.359, -56.394, 102.83, 117.787, 60.179, -67.226]
  MoveL 1159 to (-2226.52, 337.82, -103.74) mm, rotated rx 0 ry 17.72 rz 16.38 deg; joints [-33.335, -57.091, 102.665, 117.159, 59.6, -66.948]
  MoveL 1160 to (-2226.52, 317.25, -101.83) mm, rotated rx 0 ry 17.83 rz 17.21 deg; joints [-33.311, -57.749, 102.485, 116.503, 59.016, -66.761]
  MoveL 1161 to (-2226.52, 297.66, -99.91) mm, rotated rx 0 ry 17.95 rz 18.15 deg; joints [-33.286, -58.373, 102.291, 115.813, 58.423, -66.667]
  MoveL 1162 to (-2226.52, 279, -97.97) mm, rotated rx 0 ry 18.09 rz 19.21 deg; joints [-33.26, -58.965, 102.085, 115.084, 57.818, -66.673]
  MoveL 1163 to (-2226.52, 261.26, -96) mm, rotated rx 0 ry 18.25 rz 20.39 deg; joints [-33.233, -59.526, 101.866, 114.312, 57.197, -66.781]
  MoveL 1164 to (-2226.52, 244.4, -94) mm, rotated rx 0 ry 18.43 rz 21.71 deg; joints [-33.204, -60.059, 101.635, 113.489, 56.557, -66.994]
  MoveL 1165 to (-2226.52, 228.39, -91.95) mm, rotated rx 0 ry 18.64 rz 23.17 deg; joints [-33.173, -60.567, 101.392, 112.607, 55.894, -67.313]
  MoveL 1166 to (-2226.52, 213.2, -89.86) mm, rotated rx 0 ry 18.88 rz 24.79 deg; joints [-33.139, -61.05, 101.137, 111.656, 55.203, -67.737]
  MoveL 1167 to (-2226.52, 198.8, -87.71) mm, rotated rx 0 ry 19.15 rz 26.56 deg; joints [-33.102, -61.513, 100.869, 110.627, 54.48, -68.262]
  MoveL 1168 to (-2226.52, 185.15, -85.5) mm, rotated rx 0 ry 19.48 rz 28.51 deg; joints [-33.061, -61.955, 100.587, 109.506, 53.722, -68.881]
  MoveL 1169 to (-2226.52, 172.23, -83.22) mm, rotated rx 0 ry 19.86 rz 30.62 deg; joints [-33.016, -62.38, 100.291, 108.28, 52.924, -69.582]
  MoveL 1170 to (-2226.52, 160.01, -80.87) mm, rotated rx 0 ry 20.3 rz 32.9 deg; joints [-32.966, -62.789, 99.978, 106.932, 52.085, -70.347]
  MoveL 1171 to (-2226.52, 148.45, -78.44) mm, rotated rx 0 ry 20.81 rz 35.33 deg; joints [-32.909, -63.183, 99.648, 105.445, 51.201, -71.152]
  MoveL 1172 to (-2226.52, 137.53, -75.93) mm, rotated rx 0 ry 21.41 rz 37.92 deg; joints [-32.845, -63.563, 99.297, 103.797, 50.272, -71.964]
  MoveL 1173 to (-2226.52, 127.2, -73.32) mm, rotated rx 0 ry 22.11 rz 40.65 deg; joints [-32.773, -63.929, 98.924, 101.966, 49.3, -72.743]
  MoveL 1174 to (-2226.52, 127.2, -73.32) mm, rotated rx 0 ry 22.11 rz 40.65 deg; joints [-32.773, -63.929, 98.924, 101.966, 49.3, -72.743]
  MoveL 1175 to (-2226.74, 122.02, -71.85) mm, rotated rx 0 ry 22.52 rz 42.11 deg; joints [-32.735, -64.109, 98.709, 100.921, 48.779, -73.112]
  MoveL 1176 to (-2227.43, 116.94, -70.19) mm, rotated rx 0 ry 22.97 rz 43.61 deg; joints [-32.702, -64.273, 98.465, 99.798, 48.254, -73.435]
  MoveL 1177 to (-2228.6, 112.02, -68.36) mm, rotated rx 0 ry 23.45 rz 45.1 deg; joints [-32.673, -64.417, 98.192, 98.605, 47.733, -73.697]
  MoveL 1178 to (-2230.27, 107.31, -66.36) mm, rotated rx 0 ry 23.95 rz 46.57 deg; joints [-32.651, -64.539, 97.893, 97.363, 47.23, -73.887]
  MoveL 1179 to (-2232.44, 102.9, -64.24) mm, rotated rx 0 ry 24.46 rz 47.96 deg; joints [-32.636, -64.634, 97.575, 96.106, 46.76, -73.998]
  MoveL 1180 to (-2235.13, 98.84, -62.03) mm, rotated rx 0 ry 24.96 rz 49.26 deg; joints [-32.629, -64.7, 97.242, 94.862, 46.335, -74.028]
  MoveL 1181 to (-2238.32, 95.17, -59.74) mm, rotated rx 0 ry 25.44 rz 50.42 deg; joints [-32.633, -64.734, 96.898, 93.669, 45.967, -73.982]
  MoveL 1182 to (-2241.96, 91.98, -57.45) mm, rotated rx 0 ry 25.87 rz 51.41 deg; joints [-32.649, -64.735, 96.556, 92.582, 45.671, -73.874]
  MoveL 1183 to (-2246.01, 89.31, -55.2) mm, rotated rx 0 ry 26.24 rz 52.2 deg; joints [-32.677, -64.702, 96.222, 91.641, 45.454, -73.719]
  MoveL 1184 to (-2250.44, 87.18, -53.02) mm, rotated rx 0 ry 26.53 rz 52.77 deg; joints [-32.719, -64.637, 95.903, 90.876, 45.319, -73.534]
  MoveL 1185 to (-2255.15, 85.62, -50.97) mm, rotated rx 0 ry 26.73 rz 53.13 deg; joints [-32.775, -64.54, 95.607, 90.319, 45.27, -73.335]
  MoveL 1186 to (-2260.09, 84.65, -49.09) mm, rotated rx 0 ry 26.83 rz 53.25 deg; joints [-32.844, -64.415, 95.339, 89.984, 45.303, -73.134]
  MoveL 1187 to (-2265.19, 84.27, -47.39) mm, rotated rx 0 ry 26.83 rz 53.15 deg; joints [-32.925, -64.264, 95.102, 89.871, 45.416, -72.937]
  MoveL 1188 to (-2270.36, 84.46, -45.89) mm, rotated rx 0 ry 26.74 rz 52.85 deg; joints [-33.016, -64.09, 94.899, 89.972, 45.601, -72.744]
  MoveL 1189 to (-2275.55, 85.21, -44.61) mm, rotated rx 0 ry 26.57 rz 52.34 deg; joints [-33.116, -63.897, 94.729, 90.268, 45.853, -72.55]
  MoveL 1190 to (-2280.67, 86.51, -43.55) mm, rotated rx 0 ry 26.33 rz 51.65 deg; joints [-33.223, -63.687, 94.592, 90.734, 46.162, -72.35]
  MoveL 1191 to (-2285.69, 88.31, -42.7) mm, rotated rx 0 ry 26.03 rz 50.81 deg; joints [-33.333, -63.464, 94.486, 91.34, 46.521, -72.134]
  MoveL 1192 to (-2290.53, 90.6, -42.05) mm, rotated rx 0 ry 25.68 rz 49.83 deg; joints [-33.446, -63.23, 94.409, 92.058, 46.922, -71.897]
  MoveL 1193 to (-2295.17, 93.32, -41.59) mm, rotated rx 0 ry 25.31 rz 48.74 deg; joints [-33.558, -62.989, 94.357, 92.856, 47.354, -71.632]
  MoveL 1194 to (-2299.55, 96.45, -41.31) mm, rotated rx 0 ry 24.92 rz 47.57 deg; joints [-33.667, -62.744, 94.329, 93.708, 47.809, -71.337]
  MoveL 1195 to (-2307.49, 103.77, -41.23) mm, rotated rx 0 ry 24.12 rz 45.03 deg; joints [-33.875, -62.247, 94.333, 95.495, 48.76, -70.657]
  MoveL 1196 to (-2314.16, 112.28, -41.69) mm, rotated rx 0 ry 23.36 rz 42.4 deg; joints [-34.059, -61.757, 94.404, 97.279, 49.721, -69.882]
  MoveL 1197 to (-2319.46, 121.69, -42.62) mm, rotated rx 0 ry 22.67 rz 39.79 deg; joints [-34.216, -61.287, 94.531, 98.98, 50.649, -69.062]
  MoveL 1198 to (-2323.34, 131.74, -43.95) mm, rotated rx 0 ry 22.06 rz 37.29 deg; joints [-34.343, -60.847, 94.708, 100.56, 51.52, -68.251]
  MoveL 1199 to (-2325.71, 142.21, -45.65) mm, rotated rx 0 ry 21.53 rz 34.98 deg; joints [-34.439, -60.447, 94.932, 102.006, 52.317, -67.498]
  MoveL 1200 to (-2326.52, 152.83, -47.7) mm, rotated rx 0 ry 21.08 rz 32.88 deg; joints [-34.503, -60.094, 95.204, 103.321, 53.031, -66.84]
  MoveL 1201 to (-2326.52, 152.83, -47.7) mm, rotated rx 0 ry 21.08 rz 32.88 deg; joints [-34.503, -60.094, 95.204, 103.321, 53.031, -66.84]
  MoveL 1202 to (-2326.52, 173.7, -51.77) mm, rotated rx 0 ry 20.38 rz 29.36 deg; joints [-34.587, -59.459, 95.737, 105.513, 54.249, -65.769]
  MoveL 1203 to (-2326.52, 196.39, -55.63) mm, rotated rx 0 ry 19.83 rz 26.25 deg; joints [-34.657, -58.78, 96.227, 107.411, 55.374, -64.872]
  MoveL 1204 to (-2326.52, 221, -59.32) mm, rotated rx 0 ry 19.39 rz 23.55 deg; joints [-34.718, -58.05, 96.679, 109.073, 56.418, -64.199]
  MoveL 1205 to (-2326.52, 234.06, -61.1) mm, rotated rx 0 ry 19.2 rz 22.35 deg; joints [-34.746, -57.664, 96.891, 109.829, 56.914, -63.955]
  MoveL 1206 to (-2326.52, 247.64, -62.85) mm, rotated rx 0 ry 19.04 rz 21.24 deg; joints [-34.771, -57.263, 97.095, 110.543, 57.394, -63.774]
  MoveL 1207 to (-2326.52, 261.76, -64.56) mm, rotated rx 0 ry 18.89 rz 20.22 deg; joints [-34.796, -56.845, 97.29, 111.218, 57.862, -63.657]
  MoveL 1208 to (-2326.52, 276.44, -66.25) mm, rotated rx 0 ry 18.75 rz 19.28 deg; joints [-34.819, -56.411, 97.477, 111.859, 58.317, -63.603]
  MoveL 1209 to (-2326.52, 291.68, -67.92) mm, rotated rx 0 ry 18.63 rz 18.42 deg; joints [-34.842, -55.957, 97.654, 112.47, 58.762, -63.61]
  MoveL 1210 to (-2326.52, 307.5, -69.56) mm, rotated rx 0 ry 18.52 rz 17.64 deg; joints [-34.863, -55.484, 97.823, 113.052, 59.2, -63.677]
  MoveL 1211 to (-2326.52, 323.91, -71.19) mm, rotated rx 0 ry 18.42 rz 16.93 deg; joints [-34.884, -54.991, 97.982, 113.61, 59.63, -63.802]
  MoveL 1212 to (-2326.52, 340.94, -72.8) mm, rotated rx 0 ry 18.32 rz 16.28 deg; joints [-34.905, -54.476, 98.132, 114.145, 60.055, -63.984]
  MoveL 1213 to (-2326.52, 358.59, -74.41) mm, rotated rx 0 ry 18.24 rz 15.69 deg; joints [-34.924, -53.939, 98.271, 114.661, 60.477, -64.219]
  MoveL 1214 to (-2326.52, 376.87, -76.01) mm, rotated rx 0 ry 18.16 rz 15.16 deg; joints [-34.944, -53.377, 98.4, 115.157, 60.896, -64.505]
  MoveL 1215 to (-2326.52, 376.87, -76.01) mm, rotated rx 0 ry 18.16 rz 15.16 deg; joints [-34.944, -53.377, 98.4, 115.157, 60.896, -64.505]
  MoveL 1216 to (-2327.36, 389.01, -76.77) mm, rotated rx 0 ry 18.12 rz 14.85 deg; joints [-34.969, -52.981, 98.437, 115.443, 61.167, -64.691]
  MoveL 1217 to (-2329.77, 400.96, -77) mm, rotated rx 0 ry 18.09 rz 14.57 deg; joints [-35.017, -52.55, 98.393, 115.663, 61.432, -64.839]
  MoveL 1218 to (-2333.6, 412.43, -76.72) mm, rotated rx 0 ry 18.08 rz 14.32 deg; joints [-35.086, -52.098, 98.273, 115.817, 61.682, -64.946]
  MoveL 1219 to (-2338.75, 423.25, -75.96) mm, rotated rx 0 ry 18.07 rz 14.11 deg; joints [-35.174, -51.633, 98.082, 115.907, 61.915, -65.009]
  MoveL 1220 to (-2345.15, 433.21, -74.72) mm, rotated rx 0 ry 18.08 rz 13.92 deg; joints [-35.279, -51.164, 97.824, 115.932, 62.128, -65.022]
  MoveL 1221 to (-2352.74, 442.07, -73.01) mm, rotated rx 0 ry 18.11 rz 13.77 deg; joints [-35.4, -50.7, 97.499, 115.891, 62.314, -64.978]
  MoveL 1222 to (-2356.98, 446, -71.96) mm, rotated rx 0 ry 18.12 rz 13.71 deg; joints [-35.466, -50.474, 97.312, 115.845, 62.397, -64.932]
  MoveL 1223 to (-2361.49, 449.52, -70.8) mm, rotated rx 0 ry 18.14 rz 13.65 deg; joints [-35.536, -50.253, 97.109, 115.782, 62.471, -64.869]
  MoveL 1224 to (-2366.26, 452.57, -69.52) mm, rotated rx 0 ry 18.16 rz 13.61 deg; joints [-35.608, -50.041, 96.891, 115.7, 62.535, -64.788]
  MoveL 1225 to (-2371.26, 455.08, -68.12) mm, rotated rx 0 ry 18.18 rz 13.57 deg; joints [-35.684, -49.84, 96.659, 115.6, 62.589, -64.687]
  MoveL 1226 to (-2376.44, 456.98, -66.61) mm, rotated rx 0 ry 18.21 rz 13.54 deg; joints [-35.761, -49.653, 96.415, 115.482, 62.632, -64.566]
  MoveL 1227 to (-2381.77, 458.2, -65) mm, rotated rx 0 ry 18.24 rz 13.52 deg; joints [-35.839, -49.484, 96.161, 115.346, 62.662, -64.425]
  MoveL 1228 to (-2387.15, 458.67, -63.31) mm, rotated rx 0 ry 18.27 rz 13.52 deg; joints [-35.918, -49.336, 95.901, 115.193, 62.678, -64.265]
  MoveL 1229 to (-2392.46, 458.33, -61.57) mm, rotated rx 0 ry 18.31 rz 13.53 deg; joints [-35.994, -49.215, 95.641, 115.025, 62.679, -64.088]
  MoveL 1230 to (-2397.64, 457.16, -59.81) mm, rotated rx 0 ry 18.34 rz 13.54 deg; joints [-36.067, -49.122, 95.383, 114.845, 62.665, -63.897]
  MoveL 1231 to (-2402.55, 455.18, -58.08) mm, rotated rx 0 ry 18.38 rz 13.58 deg; joints [-36.135, -49.06, 95.134, 114.656, 62.637, -63.696]
  MoveL 1232 to (-2407.1, 452.43, -56.39) mm, rotated rx 0 ry 18.42 rz 13.62 deg; joints [-36.197, -49.029, 94.9, 114.462, 62.595, -63.489]
  MoveL 1233 to (-2411.22, 449.01, -54.79) mm, rotated rx 0 ry 18.45 rz 13.68 deg; joints [-36.252, -49.03, 94.684, 114.267, 62.54, -63.282]
  MoveL 1234 to (-2414.82, 445.04, -53.31) mm, rotated rx 0 ry 18.49 rz 13.75 deg; joints [-36.299, -49.059, 94.49, 114.075, 62.475, -63.081]
  MoveL 1235 to (-2417.9, 440.62, -51.95) mm, rotated rx 0 ry 18.52 rz 13.83 deg; joints [-36.339, -49.114, 94.318, 113.887, 62.401, -62.887]
  MoveL 1236 to (-2420.52, 435.76, -50.71) mm, rotated rx 0 ry 18.55 rz 13.91 deg; joints [-36.371, -49.194, 94.166, 113.702, 62.319, -62.7]
  MoveL 1237 to (-2422.69, 430.47, -49.57) mm, rotated rx 0 ry 18.58 rz 14.01 deg; joints [-36.396, -49.297, 94.034, 113.52, 62.227, -62.52]
  MoveL 1238 to (-2424.38, 424.79, -48.55) mm, rotated rx 0 ry 18.61 rz 14.12 deg; joints [-36.414, -49.423, 93.923, 113.342, 62.127, -62.349]
  MoveL 1239 to (-2425.59, 418.8, -47.67) mm, rotated rx 0 ry 18.64 rz 14.24 deg; joints [-36.425, -49.57, 93.832, 113.168, 62.02, -62.19]
  MoveL 1240 to (-2426.29, 412.7, -46.93) mm, rotated rx 0 ry 18.67 rz 14.37 deg; joints [-36.429, -49.733, 93.765, 113.005, 61.908, -62.048]
  MoveL 1241 to (-2426.52, 406.55, -46.33) mm, rotated rx 0 ry 18.69 rz 14.5 deg; joints [-36.426, -49.909, 93.719, 112.851, 61.793, -61.922]
  MoveL 1242 to (-2426.52, 406.55, -46.33) mm, rotated rx 0 ry 18.69 rz 14.5 deg; joints [-36.426, -49.909, 93.719, 112.851, 61.793, -61.922]
  MoveL 1243 to (-2426.52, 376.03, -43.68) mm, rotated rx 0 ry 18.81 rz 15.26 deg; joints [-36.393, -50.803, 93.526, 112.077, 61.201, -61.382]
  MoveL 1244 to (-2426.52, 347.17, -41.01) mm, rotated rx 0 ry 18.95 rz 16.14 deg; joints [-36.361, -51.637, 93.303, 111.26, 60.606, -60.957]
  MoveL 1245 to (-2426.52, 319.9, -38.31) mm, rotated rx 0 ry 19.11 rz 17.16 deg; joints [-36.327, -52.414, 93.053, 110.392, 60.004, -60.654]
  MoveL 1246 to (-2426.52, 294.16, -35.58) mm, rotated rx 0 ry 19.3 rz 18.33 deg; joints [-36.292, -53.138, 92.777, 109.465, 59.392, -60.48]
  Set speed (200.0 mm/s)
  MoveL 1247 to (-2426.52, 294.16, -35.58) mm, rotated rx 0 ry 19.3 rz 18.33 deg; joints [-36.292, -53.138, 92.777, 109.465, 59.392, -60.48]
  MoveC 1248 to (-2428.8, 207.06, -33.28) mm, rotated rx 0 ry 19.3 rz 18.33 deg; joints [-36.302, -55.407, 92.069, 107.757, 58.449, -57.183] to (-2435.77, 121.03, -45.39) mm, rotated rx 0 ry 19.3 rz 18.33 deg; joints [-36.583, -57.795, 91.64, 105.877, 57.854, -53.93]
  MoveL 1249 to (-2498.51, 100.24, -234.15) mm, rotated rx 0 ry 19.3 rz 18.33 deg; joints [-40.318, -62.069, 97.417, 104.142, 61.212, -54.691]
  Call PolishOff
